// TIA Portal project "Tunel_Perozovodsk_2000_V3(LowSensorWater)" (V16)

(* hardware
DEVICE "S7-1200 station_1"  S7-1200 Station
   slot 0: "Rack_0"  S7-1200 Rack  Rack  V1.0
   slot 1: "PLC_Start"  CPU 1214C DC/DC/Rly  6ES7 214-1HG40-0XB0  V4.4
   slot 2: "DI 16x24VDC_1"  SM 1221 DI16 x 24VDC  6ES7 221-1BH30-0XB0  V1.0
   slot 3: "DQ 16xRelay_1"  SM 1222 DQ16 x relay  6ES7 222-1HH32-0XB0  V2.0
   slot 4: "AI 8xRTD_1"  SM 1231 AI8 x RTD  6ES7 231-5PF32-0XB0  V2.0
   slot 5: "AQ 4x14BIT_1"  6ES7 232-4HD32-0XB0  V2.1
   slot 6: "AQ 4x14BIT_2"  6ES7 232-4HD32-0XB0  V2.1
*)

// ===== PLC "PLC_Start"  CPU 1214C DC/DC/Rly =====

VAR_GLOBAL   // PLC tag table "Default tag table"
   "rAlarm_SetMinPressSteam" AT %MW12 : Int;   // Уставка минимального давления пара
   "rAI_Press1" AT %MW14 : Int;   // Давление датчика
   "bAlarmPress1" AT %M16.0 : Bool;
   "rAlarm_SetMinPressWater" AT %MW18 : Int;   // Уставка аварийного давления воды
   "rAI_Press2" AT %MW20 : Int;
   "test_PID_P_Backup" AT %MD28 : Real;
   "testLoadBackUp" AT %M1.1 : Bool;
   "Test_eee" AT %M1.2 : Bool;
END_VAR

VAR_GLOBAL   // PLC tag table "HMI_"
   "bHMI_button_Start" AT %M2.0 : Bool;   // Кнопка старт
   "bHMI_button_Stop" AT %M2.1 : Bool;   // Кнопка стоп
   "bHMI_button_Pause" AT %M2.2 : Bool;   // Кнопка пауза
   "bHMI_Button_ConveyorStart" AT %M2.4 : Bool;   // Кнопка подтверждения старта конвейера
   "bStartAllowed" AT %M100.0 : Bool;   // Готовность к старту
   "bOpenWindStartConveyor" AT %M100.1 : Bool;   // Вызов окна подтверждения оператором старта конвейера
   "iHMI_Num_StatrPaster" AT %MW4 : Int;   // Статус работы пастризаора
   "sHMI_Text_State" AT %MB3 : Char;   // Ткстом статус пастеризатора
   "bTypePID_Zone1" AT %M8.0 : Bool;   // Тип ПИД - 1 - Охлаждение, 0 - Нагрев
   "bTypePID_Zone2" AT %M8.1 : Bool;   // Тип ПИД - 1 - Охлаждение, 0 - Нагрев
   "bTypePID_Zone3" AT %M8.2 : Bool;   // Тип ПИД - 1 - Охлаждение, 0 - Нагрев
   "bTypePID_Zone4" AT %M8.3 : Bool;   // Тип ПИД - 1 - Охлаждение, 0 - Нагрев
   "bTypePID_Zone5" AT %M8.4 : Bool;   // Тип ПИД - 1 - Охлаждение, 0 - Нагрев
   "rHMI_SpeedConveyor" AT %MD60 : Real;   // Скорость конвейера
   "rHMI_TimeHoldMin" AT %MD56 : Real;   // Для удобства восприятия времени выдержки
   "bResetCommon" AT %M0.3 : Bool;   // Глобальный сброс аварий
   "bAllAuto" AT %M0.6 : Bool;   // Перевод всего оборудования в авто с ручного
   "bZoomerOff" AT %M0.7 : Bool;   // Выкл пищалка
   "bHMI_button_Start_Sterilization" AT %M2.5 : Bool;   // Кнопка старт Стерилизации
   "bHMI_Steril_Fimish" AT %M8.7 : Bool;   // Стерилизация готова флаг
   "iHMI_Steril_sec" AT %MW22 : Int;   // СЕК таймера стерилизациии
   "iHMI_Steril_min" AT %MW26 : Int;   // МИН таймера стерилизации
   "iHMIWind_FinishStiril" AT %MW32 : Int;   // Всплывающее окно на панели
   "bOpenWindSterilFinish" AT %M34.0 : Bool;   // Вызвать окно окончание стирилизации
END_VAR

VAR_GLOBAL   // PLC tag table "DI"
   "+Кнопка экстренной остановки E-Stop №1" AT %I0.0 : Bool;
   "+Кнопка экстренной остановки E-Stop №2" AT %I0.1 : Bool;
   "+Кнопка экстренной остановки E-Stop №3" AT %I0.2 : Bool;
   "+Реле напряжения и фаз. Напряжение в норма" AT %I3.0 : Bool;
   "+Датчик уровня 1 – нижний уровень" AT %I3.1 : Bool;
   "+Датчик уровня 1 – верхний уровень" AT %I3.2 : Bool;
   "+Индуктивный датчик конвейера 1" AT %I3.3 : Bool;
   "+Преобразователь частоты готов (работа) 1" AT %I3.4 : Bool;
   "+Преобразователь частоты готов (работа) 2" AT %I3.5 : Bool;
   "+Преобразователь частоты готов (работа) 3" AT %I3.6 : Bool;
   "+Мотор-автомат 1" AT %I0.3 : Bool;
   "+Мотор-автомат 2" AT %I0.4 : Bool;
   "Мотор-автомат 3" AT %I0.5 : Bool;
   "Мотор-автомат 4" AT %I0.6 : Bool;
   "Мотор-автомат 5" AT %I0.7 : Bool;
   "Мотор-автомат 6" AT %I1.0 : Bool;
   "Мотор-автомат 7" AT %I1.1 : Bool;
   "Мотор-автомат 8" AT %I1.2 : Bool;
   "+Мотор-автомат 9" AT %I1.3 : Bool;
   "+Мотор-автомат 10" AT %I1.4 : Bool;
   "+Пускатель включен 1" AT %I2.0 : Bool;
   "Пускатель включен 2" AT %I2.1 : Bool;
   "Пускатель включен 3" AT %I2.2 : Bool;
   "Пускатель включен 4" AT %I2.3 : Bool;
   "Пускатель включен 5" AT %I2.4 : Bool;
   "Пускатель включен 6" AT %I2.5 : Bool;
   "+Мотор-автомат 11" AT %I1.5 : Bool;
   "Пускатель включен 7" AT %I2.6 : Bool;
   "+Пускатель включен 8" AT %I2.7 : Bool;
END_VAR

VAR_GLOBAL   // PLC tag table "MyTags"
   "rHoldtimeMIN_Out" AT %MD52 : Real;   // Время выдержки в мин
   "Разрешение работы конвейера" AT %M0.0 : Bool;   // Команда разрешения от Глобального блока работы
   "Авария, ошибка в системе" AT %M0.1 : Bool;   // Метка ошибок или аварий
   "iNomberZoneAlarm" AT %MW6 : Int;   // Номер зоны с отклонениями
   "bMain_AlarmSystem" AT %M2.3 : Bool;   // АВария в системе (Общая)
   "bStartWork_Main_TunelPaster" AT %M1.7 : Bool;   // Старт-Работа тунельного пастеризатора (ОБЩИЙ)
   "bHasPrior_Stop" AT %M10.1 : Bool;   // Имеется маркер разрешения "СТОП - конвейер
   "bStateZones_OK" AT %M10.0 : Bool;   // Все зоны готовы к работе
   "bStartFillBac_1" AT %M0.4 : Bool;   // Ком_Наполнение бака 1
   "bStartFillBac_2" AT %M0.5 : Bool;   // Ком_Наполнение бака 2
   "AlarmPress" AT %M0.2 : Bool;   // Общая авария давления
   "bStartWork_Sterilization" AT %M2.6 : Bool;   // Старт-Работа режима стерилизации
   "bState_Stiril_Zone_OK" AT %M1.0 : Bool;   // Все зоны готовы к стерилизации
   "iNumZoneStiril_NotOk" AT %MW24 : Int;   // Номер зоны не готовые стирилизации
END_VAR

VAR_GLOBAL   // PLC tag table "Timers_CPU"
   "Time_0.1s" AT %M500.0 : Bool;
   "Time_0.2s" AT %M500.1 : Bool;
   "Time_0.4s" AT %M500.2 : Bool;
   "Time_0.5s" AT %M500.3 : Bool;
   "Time_0.8s" AT %M500.4 : Bool;
   "Time_1s" AT %M500.5 : Bool;
   "Time_1.6s" AT %M500.6 : Bool;
   "Time_2s" AT %M500.7 : Bool;
END_VAR

VAR_GLOBAL   // PLC tag table "DO"
   "Пневмо_остров клапан 1" AT %Q0.0 : Bool;
   "Пневмо_остров клапан 2" AT %Q0.1 : Bool;
   "Пневмо_остров клапан 3" AT %Q0.2 : Bool;
   "Пневмо_остров клапан 4" AT %Q0.3 : Bool;
   "Пневмо_остров клапан 5" AT %Q0.4 : Bool;
   "Пневмо_остров клапан 6" AT %Q0.5 : Bool;
   "Пневмо_остров клапан 7" AT %Q0.6 : Bool;
   "Пневмо_остров клапан 8" AT %Q0.7 : Bool;
   "Пневмо_остров клапан 9" AT %Q1.0 : Bool;
   "Пневмо_остров клапан 10" AT %Q1.1 : Bool;
   "Преобразователь частоты - пуск 1" AT %Q4.0 : Bool;   // Реле К 9
   "Преобразователь частоты - пуск 2" AT %Q4.1 : Bool;   // Реле К 10
   "Преобразователь частоты - пуск 3" AT %Q4.2 : Bool;   // Реле К 11
   "Световая колонна - зеленый" AT %Q4.6 : Bool;
   "Световая колонна - желтый" AT %Q4.5 : Bool;
   "Световая колонна - красный" AT %Q4.4 : Bool;
   "Световая колонна – звуковой сигнал" AT %Q4.7 : Bool;
   "Пускатель №1" AT %Q5.0 : Bool;
   "Пускатель №2" AT %Q5.1 : Bool;
   "Пускатель №3" AT %Q5.2 : Bool;
   "Пускатель №4" AT %Q5.3 : Bool;
   "Пускатель №5" AT %Q5.4 : Bool;
   "Пускатель №6" AT %Q5.5 : Bool;
   "Пускатель №7" AT %Q5.6 : Bool;
   "Пускатель Воздуходувка" AT %Q5.7 : Bool;
   "Пуск транспортера" AT %Q4.3 : Bool;   // Реле К 12
END_VAR

VAR_GLOBAL   // PLC tag table "AI"
   "Датчик температуры 1" AT %IW140 : Int;   // PT100
   "Датчик температуры 2" AT %IW142 : Int;   // PT100
   "Датчик температуры 3" AT %IW144 : Int;   // PT100
   "Датчик температуры 4" AT %IW146 : Int;   // PT100
   "Датчик температуры 5" AT %IW148 : Int;   // PT100
   "Датчик температуры 6" AT %IW150 : Int;   // PT100
   "Датчик температуры 7" AT %IW152 : Int;   // PT100
   "AI_0.7_" AT %IW174 : Int;   // PT100
   "AI_0.0_Датчик давления 1" AT %IW112 : Int;   // 4-20mA
   "AI_0.1_Датчик давления 2" AT %IW114 : Int;   // 4-20mA
   "AI_0.2_Датчик давления 3" AT %IW116 : Int;   // 4-20mA
   "AI_0.3_" AT %IW118 : Int;   // 4-20mA
END_VAR

VAR_GLOBAL   // PLC tag table "AO"
   "Преобразователь частоты 1" AT %QW182 : Int;
   "Преобразователь частоты 2" AT %QW184 : Int;
   "Преобразователь частоты 3" AT %QW186 : Int;
   "Преобразователь частоты 4" AT %QW190 : Int;
   "Управляемый клапан №1" AT %QW160 : Int;
   "Управляемый клапан №2" AT %QW162 : Int;
   "Управляемый клапан №3" AT %QW164 : Int;
   "Управляемый клапан №4" AT %QW166 : Int;
   "Управляемый клапан №5" AT %QW180 : Int;
END_VAR

VAR_GLOBAL   // PLC tag table "Alarms"
   "Ai_Alarm_1" AT %M50.0 : Bool;
   "Ai_Alarm_2" AT %M50.1 : Bool;
   "Ai_Alarm_3" AT %M50.2 : Bool;
   "Ai_Alarm_4" AT %M50.3 : Bool;
   "Ai_Alarm_5" AT %M50.4 : Bool;
   "Ai_Alarm_6" AT %M50.5 : Bool;
END_VAR

VAR_GLOBAL   // PLC tag table "__TEST"
   "bT_Alarm" AT %M1.3 : Bool;
   "bTOpenWind" AT %M1.4 : Bool;
   "iTestPause" AT %MW1 : Int;
   "bTZoomOff" AT %M8.5 : Bool;
END_VAR

TYPE "FV_o/c"
   STRUCT
      bOpenCmd : Bool;   // Команда открыть (автомат)
      bManualMode : Bool;   // Ручной режим (TRUE)
      bManualOpen : Bool;   // Команда открыть в ручном режиме
      bFeedbackOpen : Bool;   // Обратная связь "Открыт"
      tMaxTime : Time;   // Время на открытие
      bResetAlarm : Bool;   // Сброс аварии
      bCheckFeedback : Bool;   // Выбирается есть ли обратная связь у клапана
      bOutOpen : Bool;   // Выход на открытие клапана
      iOutState : Int;   // Выход статуса клапана
   END_STRUCT;
END_TYPE

TYPE "ZoneStatus"
   STRUCT
      bInSetpoint : Bool;   // Зона в уставке по температуре
      bOutOfRange : Bool;   // Зона вышла от уставки на > дельта
      bHasPriority : Bool;   // Зона имеет приоритет на остановку конвейера
   END_STRUCT;
END_TYPE

TYPE "Zone_Pararm"
   STRUCT
      rTemp : Real;   // Температура с датчика
      rSet : Real := 20.0;   // Уставка
      rDeltaDown : Real := 1.0;   // ДельтаНижний предел
      rDeltaUP : Real := 1.0;   // ДельтаВерхний Предел
      bPriority : Bool;   // Приоритет
      bOUT_ZoneStatus : "ZoneStatus";   // Состояние зоны_
   END_STRUCT;
END_TYPE

TYPE "FV_regul"
   STRUCT
      bHMI_ManualMode : Bool;   // Переключение режима авто/ручно (0 - А, 1 - Р)
      "bManualOpen/Close" : Bool;   // Ручн режим выход DO для клапана
      rHMI_ManualSet : Real;   // Уставка в ручном режиме (0-100)
      "bAutoOpen/Close" : Bool;   // Авто режим Сигнал DO на выход для клапана
      rAuto_Set : Real;   // Уставка в автоматическом режиме
      iOut_AO : Int;   // Сигнал на аналоговый выход
      "rHMI_Out_FV-%" : Real;   // Состояние в % (0-100)
      "bOut_DO_Open/Close" : Bool;   // Сигнал выход для DO
      bOut_State_ValveOpen : Int;   // Cтатуса - клапан открыт (1)/закрыт(0)
   END_STRUCT;
END_TYPE

TYPE "Коэф ПИД"
   STRUCT
      Set : Real;   // Уставка
      Gain : Int;   // Коэф П
      I : DInt;   // Коэф И
      D : DInt;   // Коэф Д
   END_STRUCT;
END_TYPE

TYPE "PE_Param"
   STRUCT
      rПЕ_Задан : Real;
      rДлина_Конв : Real;
      rZ_Коэф : Real := 1.393;
      rТref : Real := 60.0;
      rТемп_Мин : Real;
      rТемп_Макс : Real;
      "rСкоростьКонв_м/мин" : Real;
      rРучноеЗначТемп : Real;
      diВремяПростоя : DInt := 60000;
      bManualTemp : Bool;
   END_STRUCT;
END_TYPE

TYPE "tipe_Pumps"
   STRUCT
      bAutoMode_Work : Bool;   // автоматический режим
      bManualMode : Bool;   // Ручной режим вкл/выкл
      bManualStart : Bool;   // Старт в ручном режиме
      rManualSpeed : Real;   // Скорость в ручном режиме
      rHMI_Speed : Real;   // Выходная скороость для HMI
      bHMI_PumpRun : Bool;   // Статус работы для HMI
      bresAlarm : Bool;   // Сброс аварий
      iStatusPump : Int;   // Статус насоса
      bIn_DryRunning : Bool;   // Сигнал сухого хода
      bIn_AutomatState : Bool;   // Вход статуса состояния автоматов
      bIn_PuskatelState : Bool;   // Вход статуса состояния пускателя
      bIn_Run_Ok_State : Bool;   // Вход подтверждения старта (частотники)
   END_STRUCT;
END_TYPE

TYPE "Tipe_Conveyor"
   STRUCT
      bManualMode : Bool;   // Ручной режим вкл/выкл
      bManualStart : Bool;   // Старт в ручном режиме
      rManualSpeed : Real;   // Скорость в ручном режиме
      bresAlarm : Bool;   // Сброс аварий
      rAutoSpeed : Real;   // Автомат_Заданная скорость конвеера
      rHMI_Speed : Real;   // Выходная скороость для HMI
      bHMI_Conv_Run : Bool;   // Статус работы для HMI
      iStatusConve : Int;   // Статус конвейера
      bIn_AutomatState : Bool;   // Вход статуса состояния автоматов
      bInPuskatelState : Bool;   // Вход статуса состояния пускателя
      bInRun_Ok_State : Bool;   // Вход подтверждения старта (частотники)
   END_STRUCT;
END_TYPE

TYPE "Tipe_DI"
   STRUCT
      f_DI_out : Bool;
      "bFiltr_on/off" : Bool := true;   // Вкл/выкл фильтрацию входа
      diTime_filtr : Time := T#100ms;   // Уставка времени фильтрации
      bSimulation : Bool;   // Включение режима симуляции
      "bSim_On/Off" : Bool;   // Управление симуляцией
   END_STRUCT;
END_TYPE

TYPE "Tipe_Filling_Bac"
   STRUCT
      bManualMode : Bool;
      bManualOpen : Bool;
      diTimeCloseValve : DInt;   // Таймер задержки закрытия клапана по верхнему уровню
   END_STRUCT;
END_TYPE

TYPE "Tipe_AI"
   STRUCT
      bSimulate : Bool;   // Вкл симуляции датчика
      rSimulateValue : Real;   // Значение симуляции датчика
      rSensor_HL : Real;   // Верхний предел датчика
      rSensor_LL : Real;   // Нижний предел датчика
      bFiltr : Bool;   // Управление фильтром значений
      rAI_Value : Real;   // Значение аналогового датчика
   END_STRUCT;
END_TYPE

TYPE "tipePress"
   STRUCT
      rInPress : Real;   // Значение с датчика
      rSetpoint : Real := 2.0;   // Уставка минимального давления
      bAlarm_Press : Bool;   // Выход АВАРИЯ
   END_STRUCT;
END_TYPE

DATA_BLOCK "Test_Beep_DB"   // DB129
{ S7_Optimized_Access := 'TRUE' }
VERSION : 0.1
// stored: InstanceOfName Test_Beep
"Test_Beep"
BEGIN
END_DATA_BLOCK

// folder: AI_Signal/AI_DB/PT100

DATA_BLOCK "AI_1_(PT100)_DB"   // DB88
{ S7_Optimized_Access := 'FALSE' }
VERSION : 0.1
// stored: InstanceOfName AI_(PT100)
"AI_(PT100)"
BEGIN
END_DATA_BLOCK

DATA_BLOCK "AI_2_(PT100)_DB"   // DB89
{ S7_Optimized_Access := 'FALSE' }
VERSION : 0.1
// stored: InstanceOfName AI_(PT100)
"AI_(PT100)"
BEGIN
END_DATA_BLOCK

DATA_BLOCK "AI_3_(PT100)_DB"   // DB91
{ S7_Optimized_Access := 'FALSE' }
VERSION : 0.1
// stored: InstanceOfName AI_(PT100)
"AI_(PT100)"
BEGIN
END_DATA_BLOCK

DATA_BLOCK "AI_4_(PT100)_DB"   // DB92
{ S7_Optimized_Access := 'FALSE' }
VERSION : 0.1
// stored: InstanceOfName AI_(PT100)
"AI_(PT100)"
BEGIN
END_DATA_BLOCK

DATA_BLOCK "AI_5_(PT100)_DB"   // DB93
{ S7_Optimized_Access := 'FALSE' }
VERSION : 0.1
// stored: InstanceOfName AI_(PT100)
"AI_(PT100)"
BEGIN
END_DATA_BLOCK

DATA_BLOCK "AI_6_(PT100)_DB"   // DB112
{ S7_Optimized_Access := 'FALSE' }
VERSION : 0.1
// stored: InstanceOfName AI_(PT100)
"AI_(PT100)"
BEGIN
END_DATA_BLOCK

DATA_BLOCK "AI_7_(PT100)_DB"   // DB113
{ S7_Optimized_Access := 'FALSE' }
VERSION : 0.1
// stored: InstanceOfName AI_(PT100)
"AI_(PT100)"
BEGIN
END_DATA_BLOCK

// folder: DB-FB

DATA_BLOCK "FB_check_For_Start_DB"   // DB1
{ S7_Optimized_Access := 'FALSE' }
VERSION : 0.1
// stored: InstanceOfName FB_check_For_Start
"FB_check_For_Start"
BEGIN
END_DATA_BLOCK

DATA_BLOCK "FB_Emergency_DB"   // DB3
{ S7_Optimized_Access := 'FALSE' }
VERSION : 0.1
// stored: InstanceOfName FB_Аварии
"FB_Аварии"
BEGIN
END_DATA_BLOCK

DATA_BLOCK "FB_CheckZoneStatus_DB"   // DB11
{ S7_Optimized_Access := 'FALSE' }
VERSION : 0.1
// stored: InstanceOfName FB_CheckZoneStatus
"FB_CheckZoneStatus"
BEGIN
END_DATA_BLOCK

DATA_BLOCK "FB_Управление конвейером_DB"   // DB18
{ S7_Optimized_Access := 'FALSE' }
VERSION : 0.1
// stored: InstanceOfName FB_Управление конвейером
"FB_Управление конвейером"
BEGIN
END_DATA_BLOCK

DATA_BLOCK "FB_GlobalStateManager_DB"   // DB31
{ S7_Optimized_Access := 'FALSE' }
VERSION : 0.1
// stored: InstanceOfName FB_GlobalStateManager
"FB_GlobalStateManager"
BEGIN
END_DATA_BLOCK

DATA_BLOCK "FB_PE_Control_DB"   // DB38
{ S7_Optimized_Access := 'TRUE' }
VERSION : 0.1
// stored: InstanceOfName FB_ПЕ_Control
"FB_ПЕ_Control"
BEGIN
END_DATA_BLOCK

DATA_BLOCK "Главный блок конвейера_DB"   // DB39
{ S7_Optimized_Access := 'TRUE' }
VERSION : 0.1
// stored: InstanceOfName FB_Главный блок конвейера
"FB_Главный блок конвейера"
BEGIN
END_DATA_BLOCK

DATA_BLOCK "R_trig_All_Auto"   // DB40
{ S7_Optimized_Access := 'TRUE' }
VERSION : 0.1
// stored: InstanceOfName R_trig
"R_trig"
BEGIN
END_DATA_BLOCK

DATA_BLOCK "FB_Sterilization_CheckZoneStatus_DB"   // DB41
{ S7_Optimized_Access := 'FALSE' }
VERSION : 0.1
// stored: InstanceOfName FB_Stiril_CheckZoneStatus
"FB_Stiril_CheckZoneStatus"
BEGIN
END_DATA_BLOCK

DATA_BLOCK "FB_Steril_Timer_DB"   // DB42
{ S7_Optimized_Access := 'TRUE' }
VERSION : 0.1
// stored: InstanceOfName FB_Steril_Timer
"FB_Steril_Timer"
BEGIN
END_DATA_BLOCK

DATA_BLOCK "Вентилятор_DB"   // DB46
{ S7_Optimized_Access := 'FALSE' }
VERSION : 0.1
// stored: InstanceOfName Pump
"Pump"
BEGIN
END_DATA_BLOCK

DATA_BLOCK "FB_Mode_Paster_DB"   // DB81
{ S7_Optimized_Access := 'TRUE' }
VERSION : 0.1
// stored: InstanceOfName FB_Mode_Paster
"FB_Mode_Paster"
BEGIN
END_DATA_BLOCK

DATA_BLOCK "FB_Filling_Bac1_DB"   // DB84
{ S7_Optimized_Access := 'TRUE' }
VERSION : 0.1
// stored: InstanceOfName FB_Filling_Bac
"FB_Filling_Bac"
BEGIN
END_DATA_BLOCK

DATA_BLOCK "FB_Filling_Bac2_DB"   // DB86
{ S7_Optimized_Access := 'TRUE' }
VERSION : 0.1
// stored: InstanceOfName FB_Filling_Bac
"FB_Filling_Bac"
BEGIN
END_DATA_BLOCK

DATA_BLOCK "FB_Press_Controll_Water_DB"   // DB96
{ S7_Optimized_Access := 'TRUE' }
VERSION : 0.1
// stored: InstanceOfName FB_Press_Controll
"FB_Press_Controll"
BEGIN
END_DATA_BLOCK

DATA_BLOCK "FB_Press_Controll_Steam_DB"   // DB97
{ S7_Optimized_Access := 'TRUE' }
VERSION : 0.1
// stored: InstanceOfName FB_Press_Controll
"FB_Press_Controll"
BEGIN
END_DATA_BLOCK

DATA_BLOCK "FB_Press_Controll_Glikol_DB"   // DB98
{ S7_Optimized_Access := 'TRUE' }
VERSION : 0.1
// stored: InstanceOfName FB_Press_Controll
"FB_Press_Controll"
BEGIN
END_DATA_BLOCK

DATA_BLOCK "R_trig_DB"   // DB99
{ S7_Optimized_Access := 'TRUE' }
VERSION : 0.1
// stored: InstanceOfName R_trig
"R_trig"
BEGIN
END_DATA_BLOCK

DATA_BLOCK "R_trig_DB_Alarm_Zoomer"   // DB101
{ S7_Optimized_Access := 'TRUE' }
VERSION : 0.1
// stored: InstanceOfName R_trig
"R_trig"
BEGIN
END_DATA_BLOCK

DATA_BLOCK "FB_SVETOFOR_DB"   // DB102
{ S7_Optimized_Access := 'TRUE' }
VERSION : 0.1
// stored: InstanceOfName FB_SVETOFOR
"FB_SVETOFOR"
BEGIN
END_DATA_BLOCK

DATA_BLOCK "FB_check_For_StartSterilization_DB"   // DB103
{ S7_Optimized_Access := 'FALSE' }
VERSION : 0.1
// stored: InstanceOfName FB_check_For_Start
"FB_check_For_Start"
BEGIN
END_DATA_BLOCK

DATA_BLOCK "FB_STIRIL_Mode_DB"   // DB115
{ S7_Optimized_Access := 'TRUE' }
VERSION : 0.1
// stored: InstanceOfName FB_Mode_STIRIL
"FB_Mode_STIRIL"
BEGIN
END_DATA_BLOCK

DATA_BLOCK "R_trig_OpenWindOper"   // DB124
{ S7_Optimized_Access := 'TRUE' }
VERSION : 0.1
// stored: InstanceOfName R_trig
"R_trig"
BEGIN
END_DATA_BLOCK

DATA_BLOCK "R_trig_Puasa"   // DB125
{ S7_Optimized_Access := 'TRUE' }
VERSION : 0.1
// stored: InstanceOfName R_trig
"R_trig"
BEGIN
END_DATA_BLOCK

// folder: DI_signal/DB_DI

DATA_BLOCK "DI_EStop1"   // DB48
{ S7_Optimized_Access := 'FALSE' }
VERSION : 0.1
// stored: InstanceOfName FB_DI
"FB_DI"
BEGIN
END_DATA_BLOCK

DATA_BLOCK "DI_EStop2"   // DB49
{ S7_Optimized_Access := 'FALSE' }
VERSION : 0.1
// stored: InstanceOfName FB_DI
"FB_DI"
BEGIN
END_DATA_BLOCK

DATA_BLOCK "DI_EStop3"   // DB50
{ S7_Optimized_Access := 'FALSE' }
VERSION : 0.1
// stored: InstanceOfName FB_DI
"FB_DI"
BEGIN
END_DATA_BLOCK

DATA_BLOCK "DI_ReleVolt"   // DB51
{ S7_Optimized_Access := 'FALSE' }
VERSION : 0.1
// stored: InstanceOfName FB_DI
"FB_DI"
BEGIN
END_DATA_BLOCK

DATA_BLOCK "DI_1_Уровень_Низ"   // DB52
{ S7_Optimized_Access := 'FALSE' }
VERSION : 0.1
// stored: InstanceOfName FB_DI
"FB_DI"
BEGIN
END_DATA_BLOCK

DATA_BLOCK "DI_1_Уровень_Верх"   // DB53
{ S7_Optimized_Access := 'FALSE' }
VERSION : 0.1
// stored: InstanceOfName FB_DI
"FB_DI"
BEGIN
END_DATA_BLOCK

DATA_BLOCK "DI_2_Уровень_Низ"   // DB54
{ S7_Optimized_Access := 'FALSE' }
VERSION : 0.1
// stored: InstanceOfName FB_DI
"FB_DI"
BEGIN
END_DATA_BLOCK

DATA_BLOCK "DI_2_Уровень_Верх"   // DB55
{ S7_Optimized_Access := 'FALSE' }
VERSION : 0.1
// stored: InstanceOfName FB_DI
"FB_DI"
BEGIN
END_DATA_BLOCK

DATA_BLOCK "DI_Индуктивный датчик конв - 1"   // DB56
{ S7_Optimized_Access := 'FALSE' }
VERSION : 0.1
// stored: InstanceOfName FB_DI
"FB_DI"
BEGIN
END_DATA_BLOCK

DATA_BLOCK "DI_Индуктивный датчик конв - 2"   // DB57
{ S7_Optimized_Access := 'FALSE' }
VERSION : 0.1
// stored: InstanceOfName FB_DI
"FB_DI"
BEGIN
END_DATA_BLOCK

DATA_BLOCK "DI_Частотник_1_Готов"   // DB58
{ S7_Optimized_Access := 'FALSE' }
VERSION : 0.1
// stored: InstanceOfName FB_DI
"FB_DI"
BEGIN
END_DATA_BLOCK

DATA_BLOCK "DI_Частотник_2_Готов"   // DB59
{ S7_Optimized_Access := 'FALSE' }
VERSION : 0.1
// stored: InstanceOfName FB_DI
"FB_DI"
BEGIN
END_DATA_BLOCK

DATA_BLOCK "DI_Частотник_3_Готов"   // DB60
{ S7_Optimized_Access := 'FALSE' }
VERSION : 0.1
// stored: InstanceOfName FB_DI
"FB_DI"
BEGIN
END_DATA_BLOCK

DATA_BLOCK "DI_Частотник_4_Готов"   // DB61
{ S7_Optimized_Access := 'FALSE' }
VERSION : 0.1
// stored: InstanceOfName FB_DI
"FB_DI"
BEGIN
END_DATA_BLOCK

DATA_BLOCK "DI_Мотор-Автомат-1(вкл)"   // DB62
{ S7_Optimized_Access := 'FALSE' }
VERSION : 0.1
// stored: InstanceOfName FB_DI
"FB_DI"
BEGIN
END_DATA_BLOCK

DATA_BLOCK "DI_Мотор-Автомат-2(вкл)"   // DB63
{ S7_Optimized_Access := 'FALSE' }
VERSION : 0.1
// stored: InstanceOfName FB_DI
"FB_DI"
BEGIN
END_DATA_BLOCK

DATA_BLOCK "DI_Мотор-Автомат-3(вкл)"   // DB64
{ S7_Optimized_Access := 'FALSE' }
VERSION : 0.1
// stored: InstanceOfName FB_DI
"FB_DI"
BEGIN
END_DATA_BLOCK

DATA_BLOCK "DI_Мотор-Автомат-4(вкл)"   // DB65
{ S7_Optimized_Access := 'FALSE' }
VERSION : 0.1
// stored: InstanceOfName FB_DI
"FB_DI"
BEGIN
END_DATA_BLOCK

DATA_BLOCK "DI_Мотор-Автомат-5(вкл)"   // DB66
{ S7_Optimized_Access := 'FALSE' }
VERSION : 0.1
// stored: InstanceOfName FB_DI
"FB_DI"
BEGIN
END_DATA_BLOCK

DATA_BLOCK "DI_Мотор-Автомат-6(вкл)"   // DB67
{ S7_Optimized_Access := 'FALSE' }
VERSION : 0.1
// stored: InstanceOfName FB_DI
"FB_DI"
BEGIN
END_DATA_BLOCK

DATA_BLOCK "DI_Мотор-Автомат-7(вкл)"   // DB68
{ S7_Optimized_Access := 'FALSE' }
VERSION : 0.1
// stored: InstanceOfName FB_DI
"FB_DI"
BEGIN
END_DATA_BLOCK

DATA_BLOCK "DI_Мотор-Автомат-8(вкл)"   // DB69
{ S7_Optimized_Access := 'FALSE' }
VERSION : 0.1
// stored: InstanceOfName FB_DI
"FB_DI"
BEGIN
END_DATA_BLOCK

DATA_BLOCK "DI_Мотор-Автомат-9(вкл)"   // DB70
{ S7_Optimized_Access := 'FALSE' }
VERSION : 0.1
// stored: InstanceOfName FB_DI
"FB_DI"
BEGIN
END_DATA_BLOCK

DATA_BLOCK "DI_Мотор-Автомат-10(вкл)"   // DB71
{ S7_Optimized_Access := 'FALSE' }
VERSION : 0.1
// stored: InstanceOfName FB_DI
"FB_DI"
BEGIN
END_DATA_BLOCK

DATA_BLOCK "DI_Пускатель - 1(вкл)"   // DB72
{ S7_Optimized_Access := 'FALSE' }
VERSION : 0.1
// stored: InstanceOfName FB_DI
"FB_DI"
BEGIN
END_DATA_BLOCK

DATA_BLOCK "DI_Пускатель - 2(вкл)"   // DB73
{ S7_Optimized_Access := 'FALSE' }
VERSION : 0.1
// stored: InstanceOfName FB_DI
"FB_DI"
BEGIN
END_DATA_BLOCK

DATA_BLOCK "DI_Пускатель - 3(вкл)"   // DB74
{ S7_Optimized_Access := 'FALSE' }
VERSION : 0.1
// stored: InstanceOfName FB_DI
"FB_DI"
BEGIN
END_DATA_BLOCK

DATA_BLOCK "DI_Пускатель - 4(вкл)"   // DB75
{ S7_Optimized_Access := 'FALSE' }
VERSION : 0.1
// stored: InstanceOfName FB_DI
"FB_DI"
BEGIN
END_DATA_BLOCK

DATA_BLOCK "DI_Пускатель - 5(вкл)"   // DB76
{ S7_Optimized_Access := 'FALSE' }
VERSION : 0.1
// stored: InstanceOfName FB_DI
"FB_DI"
BEGIN
END_DATA_BLOCK

DATA_BLOCK "DI_Пускатель - 6(вкл)"   // DB77
{ S7_Optimized_Access := 'FALSE' }
VERSION : 0.1
// stored: InstanceOfName FB_DI
"FB_DI"
BEGIN
END_DATA_BLOCK

DATA_BLOCK "DI_Мотор-Автомат-11(вкл)"   // DB116
{ S7_Optimized_Access := 'FALSE' }
VERSION : 0.1
// stored: InstanceOfName FB_DI
"FB_DI"
BEGIN
END_DATA_BLOCK

DATA_BLOCK "DI_Пускатель - 7(вкл)"   // DB117
{ S7_Optimized_Access := 'FALSE' }
VERSION : 0.1
// stored: InstanceOfName FB_DI
"FB_DI"
BEGIN
END_DATA_BLOCK

DATA_BLOCK "DI_Пускатель - 8(вкл)"   // DB118
{ S7_Optimized_Access := 'FALSE' }
VERSION : 0.1
// stored: InstanceOfName FB_DI
"FB_DI"
BEGIN
END_DATA_BLOCK

// folder: System blocks/Program resources

DATA_BLOCK "IEC_Timer_0_DB"   // DB44
{ S7_Optimized_Access := 'TRUE' }
AUTHOR : Simatic
FAMILY : IEC
NAME : IEC_TMR
VERSION : 1.0
// stored: InstanceOfName IEC_TIMER
"IEC_TIMER"
BEGIN
END_DATA_BLOCK

DATA_BLOCK "IEC_Timer_0_DB_1"   // DB45
{ S7_Optimized_Access := 'TRUE' }
AUTHOR : Simatic
FAMILY : IEC
NAME : IEC_TMR
VERSION : 1.0
// stored: InstanceOfName IEC_TIMER
"IEC_TIMER"
BEGIN
END_DATA_BLOCK

DATA_BLOCK "IEC_Timer_0_DB_3"   // DB47
{ S7_Optimized_Access := 'TRUE' }
AUTHOR : Simatic
FAMILY : IEC
NAME : IEC_TMR
VERSION : 1.0
// stored: InstanceOfName IEC_TIMER
"IEC_TIMER"
BEGIN
END_DATA_BLOCK

DATA_BLOCK "IEC_Timer_0_DB_2"   // DB100
{ S7_Optimized_Access := 'TRUE' }
AUTHOR : Simatic
FAMILY : IEC
NAME : IEC_TMR
VERSION : 1.0
// stored: InstanceOfName IEC_TIMER
"IEC_TIMER"
BEGIN
END_DATA_BLOCK

DATA_BLOCK "IEC_Timer_0_DB_4"   // DB120
{ S7_Optimized_Access := 'TRUE' }
AUTHOR : Simatic
FAMILY : IEC
NAME : IEC_TMR
VERSION : 1.0
// stored: InstanceOfName IEC_TIMER
"IEC_TIMER"
BEGIN
END_DATA_BLOCK

DATA_BLOCK "IEC_Timer_0_DB_5"   // DB121
{ S7_Optimized_Access := 'TRUE' }
AUTHOR : Simatic
FAMILY : IEC
NAME : IEC_TMR
VERSION : 1.0
// stored: InstanceOfName IEC_TIMER
"IEC_TIMER"
BEGIN
END_DATA_BLOCK

DATA_BLOCK "IEC_Timer_0_DB_10"   // DB122
{ S7_Optimized_Access := 'TRUE' }
AUTHOR : Simatic
FAMILY : IEC
NAME : IEC_TMR
VERSION : 1.0
// stored: InstanceOfName IEC_TIMER
"IEC_TIMER"
BEGIN
END_DATA_BLOCK

DATA_BLOCK "IEC_Timer_0_DB_11"   // DB123
{ S7_Optimized_Access := 'TRUE' }
AUTHOR : Simatic
FAMILY : IEC
NAME : IEC_TMR
VERSION : 1.0
// stored: InstanceOfName IEC_TIMER
"IEC_TIMER"
BEGIN
END_DATA_BLOCK

// folder: Use VARs to HMI

DATA_BLOCK "DB2_HMI_SET"   // DB2
{ S7_Optimized_Access := 'FALSE' }
VERSION : 0.1
   VAR
      dwSetMinWaitGoPause : DInt := 1;   // Время ожидания при выходе за пределы уставок
      dwSetMinWaitComeToGo : DInt := 1;   // Время ожидания при возврате к уставкам
      dwSetTimeWaitToStart : DInt := 60;   // Время ожидания выхода на режим пастеризатора
      dwSetTimeWaitToSPause : DInt := 60;   // Время ожидания Нахождения в паузе
      k_PID_Zona1 : "Коэф ПИД";   // ПИД - ЗОна 1
      k_PID_Zona2 : "Коэф ПИД";   // ПИД - зона 2
      k_PID_Zona3 : "Коэф ПИД";   // ПИД - ЗОна 3
      k_PID_Zona4 : "Коэф ПИД";   // ПИД - зона 4
      k_PID_Zona7 : "Коэф ПИД";   // ПИД - ЗОна 7
      HMI_PE : "PE_Param";
      iTime_Steriliz : Int := 10;   // Время стерилизации
   END_VAR
BEGIN
   k_PID_Zona1.Gain := 1;
   k_PID_Zona1.I := 20;
   k_PID_Zona2.Gain := 1;
   k_PID_Zona2.I := 20;
   k_PID_Zona3.Gain := 1;
   k_PID_Zona3.I := 20;
   k_PID_Zona4.Gain := 1;
   k_PID_Zona4.I := 20;
   k_PID_Zona7.Gain := 1;
   k_PID_Zona7.I := 20;
   HMI_PE.rПЕ_Задан := 65.0;
   HMI_PE.rДлина_Конв := 2.1;
   HMI_PE.rТемп_Макс := 100.0;
   HMI_PE."rСкоростьКонв_м/мин" := 0.24;
   HMI_PE.diВремяПростоя := 900000;
END_DATA_BLOCK

DATA_BLOCK "FVs_o/p"   // DB6
{ S7_Optimized_Access := 'FALSE' }
VERSION : 0.1
   VAR
      FV_1 : "FV_o/c";   // Подпитка
      FV_2 : "FV_o/c";   // Пар
      FV_3 : "FV_o/c";   // Стерилизация
   END_VAR
BEGIN
END_DATA_BLOCK

DATA_BLOCK "ЗОНЫ_Параметры"   // DB15
{ S7_Optimized_Access := 'FALSE' }
VERSION : 0.1
   VAR
      Zone_1 : "Zone_Pararm";
      Zone_2 : "Zone_Pararm";
      Zone_3 : "Zone_Pararm";
      Zone_4 : "Zone_Pararm";
      Zone_5 : "Zone_Pararm";
      Zone_6 : "Zone_Pararm";
      Zone_7 : "Zone_Pararm";
   END_VAR
BEGIN
   Zone_1.rSet := 30.0;
   Zone_2.rTemp := 0.0;
   Zone_5.rTemp := 0.0;
   Zone_1.rDeltaDown := 3.0;
   Zone_2.rDeltaDown := 3.0;
   Zone_3.rDeltaDown := 3.0;
   Zone_5.rDeltaDown := 3.0;
   Zone_2.rSet := 60.0;
   Zone_5.rSet := 20.0;
   Zone_3.bPriority := true;
END_DATA_BLOCK

DATA_BLOCK "FVs_Regul"   // DB24
{ S7_Optimized_Access := 'FALSE' }
VERSION : 0.1
   VAR
      FV_Regul_1 : "FV_regul";
      FV_Regul_2 : "FV_regul";
      FV_Regul_3 : "FV_regul";
      FV_Regul_4 : "FV_regul";
      FV_Regul_7 : "FV_regul";
   END_VAR
BEGIN
END_DATA_BLOCK

DATA_BLOCK "Pumps"   // DB30
{ S7_Optimized_Access := 'FALSE' }
VERSION : 0.1
   VAR
      Pump_1 : "tipe_Pumps";
      Pump_2 : "tipe_Pumps";
      Pump_3 : "tipe_Pumps";
      Pump_4 : "tipe_Pumps";
      Pump_5 : "tipe_Pumps";
      Pump_6 : "tipe_Pumps";
      Pump_7 : "tipe_Pumps";
   END_VAR
BEGIN
END_DATA_BLOCK

DATA_BLOCK "DI"   // DB43
{ S7_Optimized_Access := 'FALSE' }
VERSION : 0.1
   VAR
      DI_0 : "Tipe_DI";
      DI_1 : "Tipe_DI";
      DI_2 : "Tipe_DI";
      DI_3 : "Tipe_DI";
      DI_4 : "Tipe_DI";
      DI_5 : "Tipe_DI";
      DI_6 : "Tipe_DI";
      DI_7 : "Tipe_DI";
      DI_8 : "Tipe_DI";
      DI_9 : "Tipe_DI";
      DI_10 : "Tipe_DI";
      DI_11 : "Tipe_DI";
      DI_12 : "Tipe_DI";
      DI_13 : "Tipe_DI";
      DI_14 : "Tipe_DI";
      DI_15 : "Tipe_DI";
      DI_16 : "Tipe_DI";
      DI_17 : "Tipe_DI";
      DI_18 : "Tipe_DI";
      DI_19 : "Tipe_DI";
      DI_20 : "Tipe_DI";
      DI_21 : "Tipe_DI";
      DI_22 : "Tipe_DI";
      DI_23 : "Tipe_DI";
      DI_24 : "Tipe_DI";
      DI_25 : "Tipe_DI";
      DI_26 : "Tipe_DI";
      DI_27 : "Tipe_DI";
      DI_28 : "Tipe_DI";
      DI_29 : "Tipe_DI";
      DI_30 : "Tipe_DI";
      DI_31 : "Tipe_DI";
   END_VAR
BEGIN
END_DATA_BLOCK

DATA_BLOCK "Conveyor"   // DB82
{ S7_Optimized_Access := 'FALSE' }
VERSION : 0.1
   VAR
      Conveyor_1 : "Tipe_Conveyor";
      Conveyor_2 : "Tipe_Conveyor";
      Conveyor_3 : "Tipe_Conveyor";
      Conveyor_4 : "Tipe_Conveyor";
   END_VAR
BEGIN
   Conveyor_1.rManualSpeed := 0.0;
   Conveyor_1.rAutoSpeed := 70.0;
   Conveyor_2.rAutoSpeed := 50.0;
   Conveyor_3.rAutoSpeed := 60.0;
   Conveyor_4.rAutoSpeed := 70.0;
END_DATA_BLOCK

DATA_BLOCK "Vent"   // DB83
{ S7_Optimized_Access := 'FALSE' }
VERSION : 0.1
   VAR
      Vent_1 : "tipe_Pumps";   // Вентилятор обдува
   END_VAR
BEGIN
END_DATA_BLOCK

DATA_BLOCK "Filling_BacLevel"   // DB85
{ S7_Optimized_Access := 'FALSE' }
VERSION : 0.1
   VAR
      "1" : "Tipe_Filling_Bac";   // 1 бак
   END_VAR
BEGIN
   "1".diTimeCloseValve := 5;
END_DATA_BLOCK

DATA_BLOCK "Alarms"   // DB87
{ S7_Optimized_Access := 'FALSE' }
VERSION : 0.1
   VAR
      Ai_Alarm : Array[1..7] of Struct   // Аварии датчиков аналоговых
         ALARM : Bool;
         RESET : Bool;
      END_STRUCT;
      Pump_Alarm : Array[1..7] of Struct   // Аварии насосов
         ALARM : Bool;
         RESET : Bool;
      END_STRUCT;
      Conveyor_Alarm : Array[1..4] of Struct   // Аварии конвейеров
         ALARM : Bool;
         RESET : Bool;
      END_STRUCT;
      Vent_Alarm : Struct   // Авария вентиляторов
         Vent_Alarm_1 : Bool;
         RESET : Bool;
      END_STRUCT;
      Avtomat_Off : Array[1..11] of Struct   // Контроль состояния вкл мотор автоматов
         ALARM : Bool;
      END_STRUCT;
      FV_Alarm : Array[1..7] of Struct   // Авария клапанов
         ALARM : Bool;
         RESET : Bool;
      END_STRUCT;
      "xE-Stop_1" : Bool;   // Авария по кнопке 1
      "xE-Stop_2" : Bool;   // Авария по кнопке 2
      "xE-Stop_3" : Bool;   // Авария по кнопке 3
      xVoltRele : Bool;   // Авария реле контроля фаз
      xSensorConveyorZator_1 : Bool;   // Авария затор на конвейере - 1
      xSensorConveyorZator_2 : Bool;   // Авария затор на конвейере - 2
      xLongPauseConv : Bool;   // Авария, долгое ожидание выхода конвейера из паузы
      xLongWaitZoneOk : Bool;   // Ааврия, долгий выход на уставки
   END_VAR
BEGIN
END_DATA_BLOCK

DATA_BLOCK "AI_DB"   // DB90
{ S7_Optimized_Access := 'FALSE' }
VERSION : 0.1
   VAR
      AI_1 : "Tipe_AI";
      AI_2 : "Tipe_AI";
      AI_3 : "Tipe_AI";
      AI_4 : "Tipe_AI";
      AI_5 : "Tipe_AI";
      AI_6 : "Tipe_AI";
      AI_7 : "Tipe_AI";
      "AI_4-20_1" : "Tipe_AI";   // Пар
      "AI_4-20_2" : "Tipe_AI";   // Вода
      "AI_4-20_3" : "Tipe_AI";   // Гликоль
   END_VAR
BEGIN
   "AI_4-20_1".rSensor_HL := 10.0;
   "AI_4-20_2".rSensor_HL := 10.0;
   "AI_4-20_3".rSensor_HL := 10.0;
   "AI_4-20_1".bFiltr := true;
   "AI_4-20_2".bFiltr := true;
   "AI_4-20_3".bFiltr := true;
   AI_1.bFiltr := true;
   AI_2.bFiltr := true;
   AI_3.bFiltr := true;
   AI_4.bFiltr := true;
   AI_5.bFiltr := true;
END_DATA_BLOCK

DATA_BLOCK "Control_Press_DB"   // DB95
{ S7_Optimized_Access := 'FALSE' }
VERSION : 0.1
   VAR
      PressWater : "tipePress";
      PressSteam : "tipePress";
      PressGlikol : "tipePress";
   END_VAR
BEGIN
   PressWater.rSetpoint := 0.0;
   PressSteam.rSetpoint := 0.0;
   PressGlikol.rSetpoint := 0.0;
END_DATA_BLOCK

DATA_BLOCK "Зоны_Стерилизации_Парам"   // DB104
{ S7_Optimized_Access := 'FALSE' }
VERSION : 0.1
   VAR
      "Steril_Zona-1" : "Zone_Pararm";   // параметры стерилизации зона-1
      "Steril_Zona-2" : "Zone_Pararm";   // параметры стерилизации зона-2
      "Steril_Zona-3" : "Zone_Pararm";   // параметры стерилизации зона-3
      "Steril_Zona-4" : "Zone_Pararm";   // параметры стерилизации зона-4
      "Steril_Zona-5" : "Zone_Pararm";   // параметры стерилизации зона-5
      "Steril_Zona-6" : "Zone_Pararm";   // параметры стерилизации зона-6
      "Steril_Zona-7" : "Zone_Pararm";   // параметры стерилизации зона-7
   END_VAR
BEGIN
END_DATA_BLOCK

DATA_BLOCK "My_VarS"   // DB119
{ S7_Optimized_Access := 'FALSE' }
VERSION : 0.1
   VAR
      b_Woter_LowLevel_T1 : Bool;   // Низкий Уровень воды Танк-1
      b_Woter_UpLewel_T1 : Bool;   // Верхний Уровень воды Танк-2
   END_VAR
BEGIN
END_DATA_BLOCK

// folder: Зоны/DB_Zone

DATA_BLOCK "FB_Zone_Control_1_DB"   // DB12
{ S7_Optimized_Access := 'FALSE' }
VERSION : 0.1
// stored: InstanceOfName FB_Zone_Control
"FB_Zone_Control"
BEGIN
END_DATA_BLOCK

DATA_BLOCK "FB_Zone_Control_2_DB"   // DB13
{ S7_Optimized_Access := 'FALSE' }
VERSION : 0.1
// stored: InstanceOfName FB_Zone_Control
"FB_Zone_Control"
BEGIN
END_DATA_BLOCK

DATA_BLOCK "FB_Zone_Control_3_DB"   // DB14
{ S7_Optimized_Access := 'FALSE' }
VERSION : 0.1
// stored: InstanceOfName FB_Zone_Control
"FB_Zone_Control"
BEGIN
END_DATA_BLOCK

DATA_BLOCK "FB_Zone_Control_4_DB"   // DB16
{ S7_Optimized_Access := 'FALSE' }
VERSION : 0.1
// stored: InstanceOfName FB_Zone_Control
"FB_Zone_Control"
BEGIN
END_DATA_BLOCK

DATA_BLOCK "FB_Zone_Control_5_DB"   // DB17
{ S7_Optimized_Access := 'FALSE' }
VERSION : 0.1
// stored: InstanceOfName FB_Zone_Control
"FB_Zone_Control"
BEGIN
END_DATA_BLOCK

DATA_BLOCK "FB_Zone_Control_7_DB"   // DB94
{ S7_Optimized_Access := 'FALSE' }
VERSION : 0.1
// stored: InstanceOfName FB_Zone_Control
"FB_Zone_Control"
BEGIN
END_DATA_BLOCK

DATA_BLOCK "FB_Zone_Control_6_DB"   // DB114
{ S7_Optimized_Access := 'FALSE' }
VERSION : 0.1
// stored: InstanceOfName FB_Zone_Control
"FB_Zone_Control"
BEGIN
END_DATA_BLOCK

// folder: Зоны/Стерилизация

DATA_BLOCK "FB_Zone_1_Control_Steriliz_DB"   // DB105
{ S7_Optimized_Access := 'FALSE' }
VERSION : 0.1
// stored: InstanceOfName FB_Zone_Control_Steriliz
"FB_Zone_Control_Steriliz"
BEGIN
END_DATA_BLOCK

DATA_BLOCK "FB_Zone_2_Control_Стерилизация_DB"   // DB106
{ S7_Optimized_Access := 'FALSE' }
VERSION : 0.1
// stored: InstanceOfName FB_Zone_Control_Steriliz
"FB_Zone_Control_Steriliz"
BEGIN
END_DATA_BLOCK

DATA_BLOCK "FB_Zone_3_Control_Стерилизация_DB"   // DB107
{ S7_Optimized_Access := 'FALSE' }
VERSION : 0.1
// stored: InstanceOfName FB_Zone_Control_Steriliz
"FB_Zone_Control_Steriliz"
BEGIN
END_DATA_BLOCK

DATA_BLOCK "FB_Zone_4_Control_Стерилизация_DB"   // DB108
{ S7_Optimized_Access := 'FALSE' }
VERSION : 0.1
// stored: InstanceOfName FB_Zone_Control_Steriliz
"FB_Zone_Control_Steriliz"
BEGIN
END_DATA_BLOCK

DATA_BLOCK "FB_Zone_5_Control_Стерилизация_DB"   // DB109
{ S7_Optimized_Access := 'FALSE' }
VERSION : 0.1
// stored: InstanceOfName FB_Zone_Control_Steriliz
"FB_Zone_Control_Steriliz"
BEGIN
END_DATA_BLOCK

DATA_BLOCK "FB_Zone_6_Control_Стерилизация_DB"   // DB110
{ S7_Optimized_Access := 'FALSE' }
VERSION : 0.1
// stored: InstanceOfName FB_Zone_Control_Steriliz
"FB_Zone_Control_Steriliz"
BEGIN
END_DATA_BLOCK

DATA_BLOCK "FB_Zone_7_Control_Стерилизация_DB"   // DB111
{ S7_Optimized_Access := 'FALSE' }
VERSION : 0.1
// stored: InstanceOfName FB_Zone_Control_Steriliz
"FB_Zone_Control_Steriliz"
BEGIN
END_DATA_BLOCK

// folder: Клапана/FV_o/C/FV_DB

DATA_BLOCK "FV_1"   // DB4
{ S7_Optimized_Access := 'FALSE' }
VERSION : 0.1
// stored: InstanceOfName Valve(c/o)
"Valve(c/o)"
BEGIN
END_DATA_BLOCK

DATA_BLOCK "FV_2"   // DB9
{ S7_Optimized_Access := 'FALSE' }
VERSION : 0.1
// stored: InstanceOfName Valve(c/o)
"Valve(c/o)"
BEGIN
END_DATA_BLOCK

DATA_BLOCK "FV_3"   // DB10
{ S7_Optimized_Access := 'FALSE' }
VERSION : 0.1
// stored: InstanceOfName Valve(c/o)
"Valve(c/o)"
BEGIN
END_DATA_BLOCK

// folder: Клапана/FV_regul/DB

DATA_BLOCK "FV_Regul_1_DB"   // DB20
{ S7_Optimized_Access := 'FALSE' }
VERSION : 0.1
// stored: InstanceOfName Valve(regul)
"Valve(regul)"
BEGIN
END_DATA_BLOCK

DATA_BLOCK "FV_Regul_2_DB"   // DB21
{ S7_Optimized_Access := 'FALSE' }
VERSION : 0.1
// stored: InstanceOfName Valve(regul)
"Valve(regul)"
BEGIN
END_DATA_BLOCK

DATA_BLOCK "FV_Regul_3_DB"   // DB22
{ S7_Optimized_Access := 'FALSE' }
VERSION : 0.1
// stored: InstanceOfName Valve(regul)
"Valve(regul)"
BEGIN
END_DATA_BLOCK

DATA_BLOCK "FV_Regul_4_DB"   // DB23
{ S7_Optimized_Access := 'FALSE' }
VERSION : 0.1
// stored: InstanceOfName Valve(regul)
"Valve(regul)"
BEGIN
END_DATA_BLOCK

DATA_BLOCK "FV_Regul_5_DB"   // DB37
{ S7_Optimized_Access := 'FALSE' }
VERSION : 0.1
// stored: InstanceOfName Valve(regul)
"Valve(regul)"
BEGIN
END_DATA_BLOCK

// folder: Конвейера/DB

DATA_BLOCK "Конвейер_1_DB"   // DB78
{ S7_Optimized_Access := 'FALSE' }
VERSION : 0.1
// stored: InstanceOfName Pump
"Pump"
BEGIN
END_DATA_BLOCK

DATA_BLOCK "Конвейер_2_DB"   // DB79
{ S7_Optimized_Access := 'FALSE' }
VERSION : 0.1
// stored: InstanceOfName Pump
"Pump"
BEGIN
END_DATA_BLOCK

DATA_BLOCK "Конвейер_3_DB"   // DB80
{ S7_Optimized_Access := 'FALSE' }
VERSION : 0.1
// stored: InstanceOfName Pump
"Pump"
BEGIN
END_DATA_BLOCK

// folder: Насосы/DB

DATA_BLOCK "Pump_6_DB"   // DB5
{ S7_Optimized_Access := 'FALSE' }
VERSION : 0.1
// stored: InstanceOfName Pump
"Pump"
BEGIN
END_DATA_BLOCK

DATA_BLOCK "Pump_7_DB"   // DB7
{ S7_Optimized_Access := 'FALSE' }
VERSION : 0.1
// stored: InstanceOfName Pump
"Pump"
BEGIN
END_DATA_BLOCK

DATA_BLOCK "Pump_1_DB"   // DB25
{ S7_Optimized_Access := 'FALSE' }
VERSION : 0.1
// stored: InstanceOfName Pump
"Pump"
BEGIN
END_DATA_BLOCK

DATA_BLOCK "Pump_2_DB"   // DB26
{ S7_Optimized_Access := 'FALSE' }
VERSION : 0.1
// stored: InstanceOfName Pump
"Pump"
BEGIN
END_DATA_BLOCK

DATA_BLOCK "Pump_5_DB"   // DB27
{ S7_Optimized_Access := 'FALSE' }
VERSION : 0.1
// stored: InstanceOfName Pump
"Pump"
BEGIN
END_DATA_BLOCK

DATA_BLOCK "Pump_4_DB"   // DB28
{ S7_Optimized_Access := 'FALSE' }
VERSION : 0.1
// stored: InstanceOfName Pump
"Pump"
BEGIN
END_DATA_BLOCK

DATA_BLOCK "Pump_3_DB"   // DB29
{ S7_Optimized_Access := 'FALSE' }
VERSION : 0.1
// stored: InstanceOfName Pump
"Pump"
BEGIN
END_DATA_BLOCK

// folder: (top level)

FUNCTION_BLOCK "Pump"   // FB1, SCL
{ S7_Optimized_Access := 'FALSE' }
VERSION : 0.1
   VAR_INPUT
      bManualMode : Bool;   // Выбор ручного режима
      bManualStart : Bool;   // Ручной режим - старт
      bManualStop : Bool;   // Ручной режим - стоп
      rManualSpeed : Real;   // Ручной режим - скорость
      bDryRunn : Bool;   // Защита от сухого хода
      bAutoSTop : Bool;   // Остановка насоса
      bAutoStartPerm : Bool;   // Команда на работоу в авто режиме
      rAutoSpeed : Real;   // Скорость в авто режиме
      bАвтоматы : Bool;   // Готовность привода (автоматы)
      bПускатели : Bool;   // Готовность Пускателя
      bDriveRunning : Bool;   // Привод в работе
      bDriveFault : Bool;   // Привод в ошибке
      rMinSpeed : Real;   // Минимальная скорость
      rMaxSpeed : Real := 100.0;   // Максимальная скорость
      bResetFault : Bool;   // Сброс аварии
   END_VAR
   VAR_OUTPUT
      bRunCmd : Bool;   // Пуск частотника
      iSpeedOut : Int;   // Скорость насоса для аналогового выхода
      "rSpeedHMI(0-100)" : Real;   // Скорость работы (0-100) для HMI
      bPumpRunning : Bool;   // Работа
      bPumpFault : Bool;   // Авария
      iStatus : Int;   // Статус (0 - стоп 1 - работа 2 - авария)
   END_VAR
   VAR
      bFaultLatch : Bool;
      bRunRequest : Bool;
      rSpeedPump : Real;   // Скорость насоса
      TON_NotStartRun : TON_TIME;   // ТАймер ожидания сигнала о запуске
      TON_NotContactRun : TON_TIME;   // ТАймер ожидания с контактора
      TON_DryRun : TON_TIME;   // Таймер сухого хода
   END_VAR
BEGIN
   (*
   // 1. Обработка аварий
   // Обработка ожидания сигнала о работе после старта
   IF #bAutoStartPerm THEN
       ;

   END_IF;
   *)

   // 1 Ручной режим
   IF #bManualMode THEN
       // Ручной режим
       IF #bManualStart AND NOT #bManualStop THEN
           #bRunRequest := TRUE;
       ELSIF #bManualStop THEN // OR NOT #bАвтоматы THEN
           #bRunRequest := FALSE;
       END_IF;
   ELSE
       // Автоматический режим
       // 
       //Обработка аварий
       //
       //Таймер ожидания останова по сухому ходу
       #TON_DryRun(IN := NOT #bDryRunn,
                   PT := t#1s);    //
       //--------------------------------------------------------------------------------------------------------
       IF #bAutoStartPerm AND NOT #bAutoSTop AND #bDryRunn THEN
           #TON_NotStartRun(IN := NOT #bDriveRunning,PT := t#5s);  //Таймер ожидания сигнала подтверждения пуска от частотника
           #TON_NotContactRun(IN := NOT #bПускатели, PT := t#10s);  //Таймер ожидания сигнала подтверждения пуска от пускателя


       ELSE
           #TON_NotStartRun(IN :=FALSE,PT := t#5s);
           #TON_NotContactRun(IN := FALSE,PT := t#5s);
       END_IF;
       #bFaultLatch := #TON_NotStartRun.Q OR #TON_NotContactRun.Q OR (#bDriveFault OR NOT #bАвтоматы) OR (NOT #bResetFault AND #bFaultLatch); //Разкоментировать если нужна будет фиксация АЛАРМА, сброс только по входу РЕСЕТ
       #bPumpFault := #bFaultLatch;

       //Старт--------------------------------
       #bRunRequest := #bAutoStartPerm AND NOT #bPumpFault AND NOT #TON_DryRun.Q;
   END_IF;

   // 3. Задание скорости
   IF #bManualMode THEN
       #"rSpeedHMI(0-100)" := LIMIT(MN := #rMinSpeed, IN := #rManualSpeed, MX := #rMaxSpeed);
   ELSE
       #"rSpeedHMI(0-100)" := LIMIT(MN := #rMinSpeed, IN := #rAutoSpeed, MX := #rMaxSpeed);
   END_IF;

   // Преобразование значения от 0-100 до 0-27648 для аналогового выхода
   #iSpeedOut := REAL_TO_INT((#"rSpeedHMI(0-100)"/ 100.0) * 27648.0);

   // 4. Выходные команды и статусы
   // Команды старт
   #bRunCmd := #bRunRequest;

   //Выход статуса для HMI
   #bPumpRunning := #bDriveRunning AND #bRunCmd AND NOT #bAutoSTop OR (#bManualStart AND #bManualMode);



   // 5. Числовой статус (для HMI/SCADA)
   IF #bFaultLatch THEN
       #iStatus := 2; // Авария
   ELSIF #bPumpRunning THEN
       #iStatus := 1; // Работа
   ELSE
       #iStatus := 0; // Стоп
   END_IF;

   IF #bAutoSTop AND NOT #bManualMode THEN
       #bRunCmd := FALSE;
   END_IF;
END_FUNCTION_BLOCK

FUNCTION_BLOCK "FB_GlobalStateManager"   // FB2, SCL
{ S7_Optimized_Access := 'FALSE' }
VERSION : 0.1
   VAR_INPUT
      bStartCmd : Bool;   // Команда на старт от HMI
      bConfirmStart : Bool;   // Подтверждение оператора
      bResetFault : Bool;   // Сброс ошибки
      bAllSetpointsReached : Bool;   // // Все температуры достигли уставок
      bNoFaults : Bool;   // Нет аварий
      tStartTimeout : Time := T#30m;   // Время за которое пастер выходит на режим
      tReadyDelay : Time := t#10s;   // Время ожидания при выходе на режим до готовности
   END_VAR
   VAR_OUTPUT
      eState : Int;   // Текущее состояние
      bConveyorEnable : Bool;   // Разрешение на работу конвейера
      bSystemReady : Bool;   // Готовность системы
      bSystemFault : Bool;   // Состояние Fault
      sStatusText : WString;   // Текст для HMI
   END_VAR
   VAR
      tonStartTimeout : TON_TIME;   // Таймер выхода на режим
      tonReadyDelay : TON_TIME;   // Таймер готовности
   END_VAR
   VAR CONSTANT
      cSTATE_IDLE : Int;
      cSTATE_CHECK : Int := 10;
      cSTATE_STARTING : Int := 20;
      cSTATE_READY_DELAY : Int := 30;
      cSTATE_READY : Int := 40;
      cSTATE_FAULT : Int := 99;
      sText1 : String := 'Waiting';
   END_VAR
BEGIN
   // Сброс таймеров при неактивных состояниях (по требованию 1)
   IF #eState <> #cSTATE_STARTING THEN
       #tonStartTimeout(IN := FALSE,
                        PT := #tStartTimeout);
   END_IF;

   IF #eState <> #cSTATE_READY_DELAY THEN
       #tonReadyDelay(IN := FALSE,
                      PT := #tReadyDelay);
   END_IF;

   // Глобальная проверка аварии (по требованию 4)
   IF NOT #bNoFaults AND #eState <> #cSTATE_FAULT THEN
       #eState := #cSTATE_FAULT;
       #bSystemFault := TRUE;
       #bConveyorEnable := FALSE; // Принудительный останов (по требованию 2)
   ELSIF NOT #bStartCmd THEN
       #eState := #cSTATE_IDLE;
   END_IF;


   REGION Основная логика

       // Основной CASE
       CASE #eState OF
           #cSTATE_IDLE:
               #bConveyorEnable := FALSE;
               IF #bStartCmd AND #bNoFaults THEN // Запрет старта при аварии
                   #eState := #cSTATE_CHECK;
               END_IF;

           #cSTATE_CHECK:
               // Проверка уже в глобальном условии, дублирование не нужно
               #eState := #cSTATE_STARTING;

           #cSTATE_STARTING:
               IF #bAllSetpointsReached THEN
                   #eState := #cSTATE_READY_DELAY;
               ELSIF #tonStartTimeout.Q THEN
                   #eState := #cSTATE_FAULT;
               END_IF;

           #cSTATE_READY_DELAY:
               IF #tonReadyDelay.Q THEN
                   #eState := #cSTATE_READY;
               END_IF;

           #cSTATE_READY:
               #bSystemReady := TRUE;
               IF #bConfirmStart THEN
                   #bConveyorEnable := TRUE;
               END_IF;

           #cSTATE_FAULT:
               #bSystemFault := TRUE;
               #bConveyorEnable := FALSE; // Гарантированный останов
               IF #bResetFault AND #bNoFaults THEN
                   #eState := #cSTATE_IDLE;
                   #bSystemFault := FALSE;
               END_IF;

           ELSE
               #eState := #cSTATE_IDLE;
       END_CASE;

   END_REGION


   // Обновление таймеров (после логики состояний!)
   #tonStartTimeout(IN := (#eState = #cSTATE_STARTING) AND NOT #bAllSetpointsReached,
                    PT := #tStartTimeout);
   #tonReadyDelay(IN := (#eState = #cSTATE_READY_DELAY),
                  PT := #tReadyDelay);
END_FUNCTION_BLOCK

FUNCTION_BLOCK "Valve(c/o)"   // FB3, SCL
{ S7_Optimized_Access := 'FALSE' }
VERSION : 0.1
   VAR_INPUT
      bAuto_OpenCmd : Bool;   // Команда открыть (автомат)
      bManualMode : Bool;   // Ручной режим (TRUE)
      bManualOpen : Bool;   // Команда открыть в ручном режиме
      bFeedbackOpen : Bool;   // Обратная связь "Открыт"
      tMaxTime : Time;   // Время на открытие
      bResetAlarm : Bool;   // Сброс аварии
      bHaveFeedback : Bool;   // Есть ли обратная связь (0 - нет, 1 есть)
   END_VAR
   VAR_OUTPUT
      bValveOpen : Bool;   // Управляющий выход
      iValveState : Int;   // 0 = Закрыт, 1 = Открыт, 2 = Авария
      bValveFault : Bool;   // Авария
   END_VAR
   VAR
      tiOpenTimer : TON_TIME;   // Таймер на открытие
      bWaitingOpen : Bool;   // Флаг ожидания открытия
      bEnableTimer : Bool;   // Флаг активации таймера
   END_VAR
BEGIN

   // Обновление таймера — всегда в одном месте, вне условий
   #tiOpenTimer(
                IN := #bEnableTimer,
                PT := #tMaxTime
   );

   // Сброс
   IF #bResetAlarm THEN
       #bValveFault := FALSE;
       #bWaitingOpen := FALSE;
       #bEnableTimer := FALSE;
   END_IF;

   // === Режим: РУЧНОЙ ===
   IF #bManualMode THEN
       #bValveOpen := #bManualOpen;
       #bValveFault := FALSE;          // Аварии в ручном режиме не учитываются
       #bEnableTimer := FALSE;
       #bWaitingOpen := FALSE;

       // === Режим: АВТО ===
   ELSE

           // Управление выходом с учетом аварии, с контролем обратной связи
        IF #bAuto_OpenCmd AND NOT #bValveFault THEN
                   #bValveOpen := TRUE;
        ELSE
                   #bValveOpen := FALSE;
               END_IF;

               //  Проверяем, есть ли контроль обратной связи
        IF #bHaveFeedback THEN
            // Контроль открытия
            IF #bAuto_OpenCmd AND NOT #bFeedbackOpen AND NOT #bValveFault THEN
                #bEnableTimer := TRUE;
                #bWaitingOpen := TRUE;
            ELSE
                #bEnableTimer := FALSE;
                ;
                IF #bFeedbackOpen THEN
                    #bWaitingOpen := FALSE;
                END_IF;
            END_IF;
        END_IF;


           // Авария
           IF #tiOpenTimer.Q AND #bWaitingOpen THEN
               #bValveFault := TRUE;
               #bWaitingOpen := FALSE;
           END_IF;

   END_IF;


   // Состояние клапана
   IF #bValveFault THEN
       #iValveState := 2;       // Авария
   ELSIF #bHaveFeedback AND #bFeedbackOpen  THEN
       #iValveState := 1;       // Открыт
   ELSIF NOT #bHaveFeedback AND (NOT #bManualMode AND #bAuto_OpenCmd) OR (#bManualOpen AND #bManualMode) THEN
       #iValveState := 1;       // Открыт 
   ELSE
       #iValveState := 0;       // Закрыт
   END_IF;
END_FUNCTION_BLOCK

FUNCTION_BLOCK "Valve(regul)"   // FB4, SCL
{ S7_Optimized_Access := 'FALSE' }
VERSION : 0.1
   VAR_INPUT
      bManualMode : Bool;   // TRUE = ручной режим, FALSE = автоматический режим
      rAutoSetpoint : Real;   // Уставка открытия клапана в % (0.0–100.0) в автомате
      "bAutoOpen/Close" : Bool;   // Выход Do в автоматическом режиме
      rManualSetpoint : Real;   // Уставка открытия клапана в % (0.0–100.0) в ручном режиме
      "bManualOpen/Close" : Bool;   // Управление выходом открыть/закрыть
   END_VAR
   VAR_OUTPUT
      iAnalogOutput : Int;   // Значение для аналогового выхода (0–27648)
      rValvePosPercent : Real;   // Текущее % открытия клапана для HMI
      bStatusValveOpen : Int;   // Статус сигнал "клапан открыт" (TRUE, если >0%)
      "bOut_Open/Close" : Bool;   // выход для открытия клапана
   END_VAR
   VAR
      rSetpointPercent : Real;   // Расчётная уставка % открытия в текущем режиме
   END_VAR
BEGIN
       // Выбор уставки в зависимости от режима
       IF #bManualMode THEN
           #rSetpointPercent := #rManualSetpoint;
           #"bOut_Open/Close" := #"bManualOpen/Close";
       ELSE
           #rSetpointPercent := #rAutoSetpoint;
           #"bOut_Open/Close" := #"bAutoOpen/Close";
       END_IF;

       // Ограничение % от 0.0 до 100.0
       IF #rSetpointPercent < 0.0 THEN
           #rSetpointPercent := 0.0;
       ELSIF #rSetpointPercent > 100.0 THEN
           #rSetpointPercent := 100.0;
       END_IF;

       // Перевод % в значение для аналогового выхода
       #iAnalogOutput := REAL_TO_INT((#rSetpointPercent / 100.0) * 27648.0);

           // Вывод значения для HMI
       #rValvePosPercent := #rSetpointPercent;

       // Статус клапана для Панели HMI
       IF #rSetpointPercent > 0.0 AND #"bOut_Open/Close" THEN
           #bStatusValveOpen := 1;
       ELSE
           #bStatusValveOpen := 0;
       END_IF;
       ;
END_FUNCTION_BLOCK

FUNCTION_BLOCK "FB_Управление конвейером"   // FB5, SCL
{ S7_Optimized_Access := 'FALSE' }
VERSION : 0.1
   VAR_INPUT
      bEnable : Bool;   // Общий флаг работы системы
      bStartCmd : Bool;   // Команда на запуск от HMI, по кнопке из окна подтверждения
      bAllZonesInSetpoint : Bool;   // Все зоны достигли уставок
      bGlobalFault : Bool;   // Авария по системе
      bZoneHasPriority : Bool;   // У зоны с отклонением есть приоритет
      dwDeltaTempDelayMin : DWord;   // Задержка (мин), прежде чем остановить конвейер при отклонении
      dwResumeDelayMin : DInt;   // Время возврата после нормализации
   END_VAR
   VAR_OUTPUT
      bConveyorRun : Bool;   // Команда на пуск частотников
      bReadyToStart : Bool;   // Готовность к работе конвейера
      bWaitingConfirm : Bool;   // Ждём подтверждения от оператора, вывод окна на HMI
      bPaused : Bool;   // Конвейер остановлен по отклонению
   END_VAR
   VAR
      bStarted : Bool;   // Внутреннее состояние — процесс стартовал
      tiPauseTimer : TON_TIME;   // Таймер задержки перед остановкой
      tiResumeTimer : TON_TIME;   // Таймер ожидания перед возобновлением
      aZoneS_Status : Array[1..5] of "ZoneStatus";   // Массив для сбора состояния зон
      i : Int;
   END_VAR
   // tiPauseTimer.PT := T#1s;
   // tiResumeTimer.PT := T#1s;
BEGIN

   // Проверка на наличие флага обей работы системы
   IF NOT #bEnable THEN
       #bReadyToStart := FALSE;
       #bWaitingConfirm := FALSE;
       #bConveyorRun := FALSE;
       #bPaused := FALSE;
       #tiPauseTimer.IN := FALSE;
       #tiResumeTimer.IN := FALSE;
       RETURN;
   END_IF;



   // Условия готовности к запуску
   IF NOT #bStarted AND NOT #bGlobalFault AND #bAllZonesInSetpoint THEN
       #bReadyToStart := TRUE;

           // Команда на старт — вручную подтверждена
           IF NOT #bStartCmd THEN
               #bWaitingConfirm := TRUE;
           END_IF;

   ELSE
       #bReadyToStart := FALSE;
       #bWaitingConfirm := FALSE;
   END_IF;



   IF #bStartCmd AND #bReadyToStart THEN
       #bStarted := TRUE;
       #bWaitingConfirm := FALSE;
   END_IF;

   // После старта разрешаем работу, если нет аварий и температур в норме
   IF #bStarted AND NOT #bGlobalFault THEN

       IF NOT #bAllZonesInSetpoint THEN
           IF #bZoneHasPriority THEN
               // Включаем таймер паузы, задержка перед остановкой
               #tiPauseTimer(IN := TRUE,
                             PT := (#dwDeltaTempDelayMin * 60000)) //В минутах
               ;
           ELSE
               #tiPauseTimer(IN := FALSE,PT := t#0s);
           END_IF;

           // Переход в паузу
           IF #tiPauseTimer.Q THEN
               #bPaused := TRUE;
               #bConveyorRun := FALSE;
               #tiResumeTimer(IN := FALSE, PT := t#0s); // Сброс таймера возобновления

           END_IF;

       ELSE
           // Температуры вернулись в норму — запускаем таймер на возврат
           IF #bPaused THEN
               #tiResumeTimer(IN := TRUE,
                              PT := (#dwResumeDelayMin * 60000)) // в минутах
               ;
               // Возвращаемся к работе
               IF #tiResumeTimer.Q THEN
                   #bPaused := FALSE;
                   #bConveyorRun := TRUE;
                   #tiResumeTimer(IN := FALSE, PT := t#0s); // сброс таймера
               END_IF;
           ELSE
               #bConveyorRun := TRUE;
               #tiPauseTimer(IN := FALSE, PT := t#0s); // сброс
               #tiResumeTimer(IN := FALSE,PT := t#0s);
           END_IF;
       END_IF;
   ELSE
       // Если глобальная авария — всё стоп
       #bConveyorRun := FALSE;
       #bPaused := FALSE;
       #bStarted := FALSE;
       #tiPauseTimer(IN := FALSE, PT := t#0s);
       #tiResumeTimer(IN := FALSE,PT := t#0s);
       #bWaitingConfirm := FALSE;
   END_IF;
END_FUNCTION_BLOCK

FUNCTION_BLOCK "FB_Motor_Conveyor"   // FB6, SCL
{ S7_Optimized_Access := 'FALSE' }
VERSION : 0.1
   VAR_INPUT
      bManualMode : Bool;   // Выбор ручного режима
      bManualStart : Bool;   // Ручной режим - старт
      bManualStop : Bool;   // Ручной режим - стоп
      rManualSpeed : Real;   // Ручной режим - скорость
      bAutoStartPerm : Bool;   // Команда на работоу в авто режиме
      rAutoSpeed : Real;   // Скорость в авто режиме
      bDriveReady : Bool;   // Готовность привода (автоматы)
      bDriveRunning : Bool;   // Привод в работе
      bDriveFault : Bool;   // Привод в ошибке
      rMinSpeed : Real;   // Минимальная скорость
      rMaxSpeed : Real;   // Максимальная скорость
      bResetFault : Bool;   // Сброс аварии
   END_VAR
   VAR_OUTPUT
      bRunCmd : Bool;   // Пуск частотника
      "rSpeedHMI(0-100)" : Real;   // Скорость работы (0-100) для HMI
      iSpeedOut : Int;   // Скорость насоса для аналогового выхода
      bPumpRunning : Bool;   // Работа
      bPumpFault : Bool;   // Авария
      iStatus : Int;   // Статус (0 - стоп 1 - работа 2 - авария)
   END_VAR
   VAR
      bFaultLatch : Bool;
      bRunRequest : Bool;
      rSpeedPump : Real;   // Скорость насоса
   END_VAR
BEGIN
   // 1. Обработка аварий
   #bFaultLatch := (#bDriveFault OR #bFaultLatch) AND NOT #bResetFault;
   #bPumpFault := #bFaultLatch;

   // 2. Формирование команды "Пуск"
   IF #bManualMode THEN
       // Ручной режим
       IF #bManualStart AND NOT #bManualStop THEN
           #bRunRequest := TRUE;
       ELSIF #bManualStop OR NOT #bDriveReady THEN
           #bRunRequest := FALSE;
       END_IF;
   ELSE
       // Автоматический режим
       #bRunRequest := #bAutoStartPerm AND NOT #bDriveFault;
   END_IF;

   // 3. Задание скорости
   IF #bManualMode THEN
       #"rSpeedHMI(0-100)" := LIMIT(MN := #rMinSpeed, IN := #rManualSpeed, MX := #rMaxSpeed);
   ELSE
       #"rSpeedHMI(0-100)" := LIMIT(MN := #rMinSpeed, IN := #rAutoSpeed, MX := #rMaxSpeed);
   END_IF;

   // Преобразование значения от 0-100 до 0-27648 для аналогового выхода
   #iSpeedOut := REAL_TO_INT((#"rSpeedHMI(0-100)"/ 100.0) * 27648.0);

   // 4. Выходные команды и статусы
   #bRunCmd := #bRunRequest AND NOT #bFaultLatch AND #bDriveReady;
   #bPumpRunning := #bDriveRunning AND #bRunCmd;

   // 5. Числовой статус (для HMI/SCADA)
   IF #bFaultLatch THEN
       #iStatus := 2; // Авария
   ELSIF #bPumpRunning THEN
       #iStatus := 1; // Работа
   ELSE
       #iStatus := 0; // Стоп
   END_IF;
END_FUNCTION_BLOCK

FUNCTION_BLOCK "FB_Аварии"   // FB7, SCL
{ S7_Optimized_Access := 'FALSE' }
VERSION : 0.1
   VAR_INPUT
      Rtrig_Reset : Bool;
   END_VAR
   VAR_OUTPUT
      ALARM_Active : Bool;   // Флаг активной аварии
   END_VAR
   VAR
      LatchedEmergency : Bool;   // Зафиксированная аварийная ситуация
      bAlarmAvtomats : Bool;   // Авария автоматов
      bAlarmAI : Bool;   // Авария аналоговых датчиков
      bAlarmPumps : Bool;   // Авария насосов
      bAlarmConveyors : Bool;   // Авария Конвейеров
      bAlarmFVs : Bool;   // Авария клапанов
      bAlarmDI_all : Bool;   // Авария по дискретным входам "общая"
      bAlarmLowLevel : Bool;   // Авария по низкому уровню емкостей
      mReset : Bool;
      TON_LowLevel : TON_TIME;   // Таймер для аварийного уровня емкостей
      bResetaALARM : Bool;   // Сброс аварии (кнопка на панели/системе)
   END_VAR
   VAR_TEMP
      nAi : Int;
      nPump : Int;
      nConv : Int;
      nFV : Int;
      nAvtomat : Int;
      numPump : Int;
   END_VAR
BEGIN
   REGION Предварительное отрицание
       // Сброс в 0 при отсутсвии аварий для цикла и массивов
       #bAlarmAvtomats := FALSE;
       #bAlarmAI := FALSE;
       #bAlarmPumps := FALSE;
       #bAlarmConveyors := FALSE;
       #bAlarmFVs := FALSE;


   END_REGION



   //Авария автоматические выключатели
   //--------------------------
   //
   "Alarms".Avtomat_Off[1].ALARM := NOT "Conveyor".Conveyor_1.bIn_AutomatState;
   "Alarms".Avtomat_Off[2].ALARM := NOT "Conveyor".Conveyor_2.bIn_AutomatState;
   "Alarms".Avtomat_Off[3].ALARM := NOT "Conveyor".Conveyor_3.bIn_AutomatState;
   "Alarms".Avtomat_Off[4].ALARM  :=  NOT "Pumps".Pump_1.bIn_AutomatState;
   "Alarms".Avtomat_Off[5].ALARM  :=  NOT "Pumps".Pump_2.bIn_AutomatState;
   "Alarms".Avtomat_Off[6].ALARM  :=  NOT "Pumps".Pump_3.bIn_AutomatState;
   "Alarms".Avtomat_Off[7].ALARM  :=  NOT "Pumps".Pump_4.bIn_AutomatState;
   "Alarms".Avtomat_Off[8].ALARM  :=  NOT "Pumps".Pump_5.bIn_AutomatState;
   "Alarms".Avtomat_Off[9].ALARM  :=  NOT "Pumps".Pump_6.bIn_AutomatState;
   "Alarms".Avtomat_Off[10].ALARM  :=  NOT "Pumps".Pump_7.bIn_AutomatState;
   "Alarms".Avtomat_Off[11].ALARM  :=  NOT "Vent".Vent_1.bIn_AutomatState;


   FOR #nAvtomat := 1 TO 11 DO
       IF "Alarms".Avtomat_Off[#nAvtomat].ALARM THEN
           #bAlarmAvtomats := TRUE;
       END_IF;
   END_FOR;

   //Авария аналоговых входов
   //--------------------------
   FOR #nAi := 1 TO 7 DO
       IF "Alarms".Ai_Alarm[#nAi].ALARM THEN
           #bAlarmAI := TRUE;
       END_IF;
   END_FOR;

   //Авария НАСОСОВ
   //--------------------------

   FOR #nPump := 1 TO 7 DO
       IF "Alarms".Pump_Alarm[#nPump].ALARM THEN
           #bAlarmPumps := TRUE;
           #numPump := #nPump;

       END_IF;
   END_FOR;

   //Авария КОНВЕЙЕРОВ
   //--------------------------

   FOR #nConv := 1 TO 4 DO
       IF "Alarms".Conveyor_Alarm[#nConv].ALARM THEN
           #bAlarmConveyors := TRUE;
       END_IF;
   END_FOR;

   //Авария Клапанов
   //--------------------------

   FOR #nFV := 1 TO 7 DO
       IF "Alarms".FV_Alarm[#nFV].ALARM THEN
           #bAlarmFVs := TRUE;
       END_IF;
   END_FOR;

   //Авария под давлению
   //--------------------------
   "AlarmPress" := "Control_Press_DB".PressWater.bAlarm_Press OR "Control_Press_DB".PressSteam.bAlarm_Press OR "Control_Press_DB".PressGlikol.bAlarm_Press;

   //Авария по нижним датчикам уровня емкостей
   //

   //#bAlarmLowLevel := NOT "My_VarS".b_Woter_LowLevel_T1;

   //Авария по входам DI
   //---------------------------

   #bAlarmDI_all :="Alarms"."xE-Stop_1" OR
                   "Alarms"."xE-Stop_2" OR
                   "Alarms"."xE-Stop_3" OR
                   "Alarms".xVoltRele OR
                   "Alarms".xSensorConveyorZator_1 OR
                  // "Alarms".xSensorConveyorZator_2 OR
                   "Alarms".xLongPauseConv OR
                   "Alarms".xLongWaitZoneOk;

   //Обработка всех аварий с выводом сигнала наличия АВАРИЯ
   //----------------------------------------------------------------
                   IF #bAlarmAvtomats OR
                       #bAlarmAI OR
                       #bAlarmPumps OR
                       #bAlarmConveyors OR
                       #bAlarmFVs OR
                       #bAlarmDI_all OR
                       #bAlarmLowLevel
                   THEN

                       #ALARM_Active := TRUE;
                   END_IF;
     (*                     
   //Отлавливаем фронт Ресета....................................

   #bResetaALARM := #Rtrig_Reset AND NOT #mReset;
   #mReset := #Rtrig_Reset;
   *)

    //Если нужен жесткий сбро, игнорирует все аварии                      
   #bResetaALARM := #Rtrig_Reset;

   //-------------------------------------------------------------                       
                          // Сброс аварии
   IF #bResetaALARM THEN
       #ALARM_Active := FALSE;
   END_IF;
END_FUNCTION_BLOCK

FUNCTION_BLOCK "FB_Zone_Control"   // FB8, SCL
{ S7_Optimized_Access := 'FALSE' }
VERSION : 0.1
   VAR_INPUT
      bNewStart : Bool;   // Обнаружение нового старта, уставка без дельты
      rTempActual : Real;   // Температура с датчика
      rTempSetpoint : Real;   // Уставка температуры
      rDeltaDown : Real;   // Верхнее Допустимое отклонение от уставки
      rDeltaUp : Real;   // Верхнее Допустимое отклонение от уставки
      bPriority : Bool;   // Приоритет управления конвейером (1 - стоп конвейер)
   END_VAR
   VAR_OUTPUT
      ZoneStatusOut : "ZoneStatus";
      bInSetpoint : Bool;
      bOutOfRange : Bool;
      bHasPriority : Bool;
   END_VAR
   VAR
      R_Trig_Start : "R_trig";
      "#bNewStartCLic" : Bool;
      bSetpointReachedOnce : Bool;
   END_VAR
BEGIN
   // --- Сброс флага при необходимости ---
   // 
       //----Отслеживание нажания старта, по верхнему фронту-----
   #R_Trig_Start("In":= #bNewStart,Q => #"#bNewStartCLic");

   IF #"#bNewStartCLic" THEN
       #bSetpointReachedOnce := FALSE;
   END_IF;

   // --- Фиксация первого достижения уставки (точно или ±0.1) ---
   IF NOT #bSetpointReachedOnce AND ABS(#rTempActual - #rTempSetpoint) <= 1 THEN
       #bSetpointReachedOnce := TRUE;
   END_IF;

   // --- Расчёт попадания в уставку с учетом асимметричной дельты ---
   IF #bSetpointReachedOnce THEN
       #ZoneStatusOut.bInSetpoint := (#rTempActual >= (#rTempSetpoint - #rDeltaDown)) AND
                                       (#rTempActual <= (#rTempSetpoint + #rDeltaUp));
   ELSE
       // До первого достижения — строгое приближение (или узкая дельта)
       #ZoneStatusOut.bInSetpoint := ABS(#rTempActual - #rTempSetpoint) <= 1;
   END_IF;

   //Контроль зоны выхода из уставок значительно, греем снова до уставки до разрешения на старт

   IF (#rTempActual < (#rTempSetpoint - #rDeltaDown)) OR
       (#rTempActual > (#rTempSetpoint + #rDeltaUp)) THEN
       #bSetpointReachedOnce := FALSE;
   END_IF;


   // --- Остальные сигналы ---
   #ZoneStatusOut.bOutOfRange := NOT #ZoneStatusOut.bInSetpoint;
   #ZoneStatusOut.bHasPriority := #bPriority;

   // Зеркалируем, если нужно
   #bInSetpoint := #ZoneStatusOut.bInSetpoint;
   #bOutOfRange := #ZoneStatusOut.bOutOfRange;
   #bHasPriority := #ZoneStatusOut.bHasPriority;
END_FUNCTION_BLOCK

FUNCTION_BLOCK "FB_check_For_Start"   // FB9, SCL
{ S7_Optimized_Access := 'FALSE' }
VERSION : 0.1
   VAR_INPUT
      xHMI_Start : Bool;   // кнопка старта с HMI
      xEmergency_Stop : Bool;   // аварийный стоп
      xSystem_Ready : Bool;   // Готовность всех систем
      xStopHMI : Bool;   // Кнопка СТОП на HMI
   END_VAR
   VAR_OUTPUT
      xStart_Allowed : Bool;   // Разрешение на РАБОТУ
      xStart : Bool;   // Работа пастеризатора
   END_VAR
   VAR
      "m" : Bool;   // memory
   END_VAR
BEGIN

   //Проверка на разрешение работы.
   //
   IF NOT #xEmergency_Stop AND #xSystem_Ready THEN
       #xStart_Allowed := TRUE;
   ELSE
       #xStart_Allowed := FALSE;
   END_IF;

   #xStart := (#xStart OR #xHMI_Start) AND NOT (#xEmergency_Stop OR #xStopHMI);
END_FUNCTION_BLOCK

FUNCTION_BLOCK "FB_Stiril_CheckZoneStatus"   // FB10, SCL
{ S7_Optimized_Access := 'FALSE' }
VERSION : 0.1
   VAR_OUTPUT
      bAllZones_Redy : Bool;   // Выход состояния всех зон ОК
      bPriority_Stop : Bool;   // Выход 1 - если есть метка остановки конвейера
      iZonesNumberFail : Int;   // ВЫход с Номером зоны
   END_VAR
   VAR
      aZoneS_Status : Array[1..7] of "ZoneStatus";   // Массив с данными по всем зонам
      i : Int;
      AllZone_Ok : Bool;   // Состояние всех зон ОК
      HaveStopPriority : Bool;   // В зоне есть метка для остановки конвейера
      iNumber : Int;   // Номер зоны, где отклонение температуры
   END_VAR
BEGIN

   //Что бы не контролировал готовность зоны 4 ее не надо контролировать
   //"ЗОНЫ_Параметры".Zone_4.bOUT_ZoneStatus.bInSetpoint := TRUE;
   //-------------------------------------------------------------------------------------------//
   //
           // ----Сбор данных по всем зонам в массив для обработки-----
           #aZoneS_Status[1] := "Зоны_Стерилизации_Парам"."Steril_Zona-1".bOUT_ZoneStatus;
           #aZoneS_Status[2] := "Зоны_Стерилизации_Парам"."Steril_Zona-2".bOUT_ZoneStatus;
           #aZoneS_Status[3] := "Зоны_Стерилизации_Парам"."Steril_Zona-3".bOUT_ZoneStatus;
           #aZoneS_Status[4] := "Зоны_Стерилизации_Парам"."Steril_Zona-4".bOUT_ZoneStatus;
           #aZoneS_Status[5] := "Зоны_Стерилизации_Парам"."Steril_Zona-5".bOUT_ZoneStatus;
           #aZoneS_Status[6] := "Зоны_Стерилизации_Парам"."Steril_Zona-6".bOUT_ZoneStatus;
           #aZoneS_Status[7] := "Зоны_Стерилизации_Парам"."Steril_Zona-7".bOUT_ZoneStatus;


           //Сброс маркеров по умолчанию----
   #AllZone_Ok := TRUE;    
   #HaveStopPriority := FALSE;
   #iNumber := 0;
              // ----Цикл для перебора всех зон значение выставить по количеству зон----
   FOR #i := 1 TO 7 DO
       IF NOT #aZoneS_Status[#i].bInSetpoint THEN
           #AllZone_Ok := FALSE;
           #iNumber := #i;
           IF #aZoneS_Status[#i].bHasPriority THEN
               #HaveStopPriority := TRUE;
           END_IF;
       END_IF;
   END_FOR;

   /// Присвоение переменных к выходам
   #bAllZones_Redy := #AllZone_Ok;
   #bPriority_Stop := #HaveStopPriority;
   #iZonesNumberFail := #iNumber;
END_FUNCTION_BLOCK

FUNCTION_BLOCK "FB_ПЕ_Control"   // FB11, SCL
{ S7_Optimized_Access := 'TRUE' }
VERSION : 0.1
   VAR_INPUT
      bRunRequest : Bool;   // Запрос на работу
      rSpeedPercent : Real;   // Заданная скорость от оператора (0…100%)
      rPESetpoint : Real;   // Заданное количество ПЕ
      rConveyorLength : Real := 8.3;   // Длина зоны выдержки, м
      rVmax : Real := 0.0085;   // Макс скорость м/мин
      rZParam : Real := 1.393;   // Коэффициент z (1.393 обычно)
      rTref : Real := 60.0;   // Базовая температура (обычно 60°C)
      rTmin : Real;   // Мин допустимая температура
      rTmax : Real := 75.0;   // Макс допустимая температура
      bManualMode : Bool;   // Режим "ручной расчёт температуры"
      rManualTemp : Real;   // Температура в ручном режиме
      tStopTolerance : Time;   // Допустимое время простоя
   END_VAR
   VAR_OUTPUT
      rTempSetpoint : Real;   // Уставка температуры
      rHoldTime : Real;   // Время выдержки в мин
      rConveyorSpeed : Real;   // Скорость конвейера (м/мин)
      rPENeededPerMin : Real;   // Требуемое ПЕ в минуту
      bTempValid : Bool;   // Температура в пределах допустимого
      bAlarmTempHigh : Bool;   // Температура превышает максимум
      bAlarmTempLow : Bool;   // Температура ниже минимума
      bStoppedTooLong : Bool;   // Превышено время простоя
      bAlarmTempOverride : Bool;   // Принудительная уставка из-за аварии
   END_VAR
   VAR RETAIN
      rSpeedRatio : Real;   // Отношение скорости
      rLogArg : Real;   // Аргумент логарифма
   END_VAR
   VAR
      TON_StopDelay : TON_TIME;   // Таймер задержки останова
   END_VAR
BEGIN
   // Блок управления уставкой температуры по ПЕ и скорости
   // Сначала сброс в случае остановки
   IF NOT #bRunRequest THEN
       //#rTempSetpoint := 0.0;
       #rHoldTime := 0.0;
       #rConveyorSpeed := 0.000;
       #bTempValid := TRUE;
       #bAlarmTempHigh:= FALSE;
       #bAlarmTempLow := FALSE;
       #bAlarmTempOverride := FALSE;
       #bStoppedTooLong := FALSE;
       #TON_StopDelay(IN := FALSE, PT := t#0s);
       //RETURN;
   END_IF;


   // Преобразуем % скорости в отношение
   #rSpeedRatio := #rSpeedPercent / 100.0;

   // Расчёт фактической скорости (м/с)
   #rConveyorSpeed := #rVmax * #rSpeedRatio;

   // Время нахождения бутылки в зоне (мин)
   IF #rConveyorSpeed > 0.0 THEN
       #rHoldTime := #rConveyorLength / #rConveyorSpeed; // В мин
   ELSE
       #rHoldTime := 0.0;
   END_IF;


   IF #bManualMode THEN
       // Ручной режим — берём температуру с панели
       #rTempSetpoint := #rManualTemp;
   ELSE
       // Расчёт температуры по ПЕ
       IF #rHoldTime > 0.0 AND #rPESetpoint > 0.0 THEN
           #rPENeededPerMin := #rPESetpoint / #rHoldTime;
           #rTempSetpoint := #rTref + (LN(#rPENeededPerMin) / LN(#rZParam));


           (*
           #rLogArg := LN(#rPENeededPerMin) / LN(10.0);
           #rTempSetpoint := #rTref + #rLogArg / #rZParam;
           *)
       ELSE
           #rTempSetpoint := #rTref; // по умолчанию
       END_IF;
   END_IF;

   // Проверка пределов
   #bTempValid := TRUE;
   #bAlarmTempHigh := FALSE;
   #bAlarmTempLow := FALSE;


   IF #rTempSetpoint > #rTmax THEN
       #rTempSetpoint := #rTmax;
       #bTempValid := FALSE;
       #bAlarmTempHigh := TRUE;
   ELSIF #rTempSetpoint < #rTmin THEN
       #rTempSetpoint := #rTmin;
       #bTempValid := FALSE;
       #bAlarmTempLow := TRUE;
   END_IF;
END_FUNCTION_BLOCK

FUNCTION_BLOCK "FB_Главный блок конвейера"   // FB12, SCL
{ S7_Optimized_Access := 'TRUE' }
VERSION : 0.1
   VAR_INPUT
      bModePaster : Bool;   // Режим пастеризации
      bModeStiril : Bool;   // Режим сетрилизации
      bAlarmSystem : Bool;   // Общая авария
      bResAlarm : Bool;   // Сброс аварий
      bStartCMD : Bool;   // Подтверждение оператором старта
      bAllZone_Ok : Bool;   // Маркер - все зоны ОК
      bHasPauseKonv : Bool;   // Маркер - пауза конвейера
      tiWaitZone : DInt;   // HMI - мин - Время ожидания выхода на режим
      tiWaitPause : DInt;   // HMI - мин - Время ожидания возврата с паузы
      tiWaitToGoPause : DInt;   // HMI-сек Время задержки для перехода на паузу
      tiWaitToCameGo : DInt;   // HMI- сек Время задержки для возврата в рабочий режим
   END_VAR
   VAR_OUTPUT
      iStep : Int;   // Шаг конвейера
      bKonveyorRun : Bool;   // Разрешение на работу конвейера
      bAlarmToLongPause : Bool;   // Авария по превышения ожидания выхода с паузы
      bAlarmToLongWaitZone_Ok : Bool;   // Авария по превышения ожидания выхода на режим
      bOpenWindOper : Bool;   // вызов окна оператора
   END_VAR
   VAR
      TON_WaitZones : TON_TIME;   // Таймер ожидания перехода в готовность, или в Аварию
      TON_PauseWait : TON_TIME;   // Таймер ожидания возврата с паузы до перехода в аварию
      TON_WaitToGoPaus : TON_TIME;   // Задержка для перехода в паузу
      TON_WaitToComeGo : TON_TIME;   // Задержка для выхода из паузу
      bAlarm_Timer : Bool;   // общий меркер по авариям внутри конве
   END_VAR
   VAR CONSTANT
      S_STOP : Int;   // Шаги
      S_Start_WaitZones : Int := 10;
      S_ConfirmStart : Int := 20;
      S_Working : Int := 30;
      S_Paused : Int := 40;
      S_Sterilization : Int := 50;
      S_Alarm : Int := 99;
      ConstMin : DInt := 60000;   // Минуты
      ConstS : DInt := 1000;   // Секунды
   END_VAR
BEGIN

   // Проверяем блок на наличие внешних аварий и наличие разрешения на работу
   #bOpenWindOper := FALSE;


   IF #bAlarmSystem OR #bAlarm_Timer THEN
       #iStep := #S_Alarm;
   ELSIF
       NOT #bModePaster AND NOT #bModeStiril AND NOT (#iStep = #S_Alarm) THEN
       #iStep := #S_STOP;
   END_IF;


   CASE #iStep OF
           //...................................................................................................................................................        
       #S_STOP: // ШАГ - СТОП 0
           //....Сбрасываем таймеры.......
           #TON_WaitToGoPaus(IN := FALSE,
                             PT := t#0s);
           #TON_WaitToComeGo(IN := FALSE,
                             PT := t#0s);
           #TON_WaitZones(IN := FALSE,
                          PT := t#0s);
           #TON_PauseWait(IN := FALSE,
                          PT := t#0s);

           #bKonveyorRun := FALSE;


           IF #bModePaster THEN
               #iStep := #S_Start_WaitZones;
           ELSIF #bModeStiril THEN
               #iStep := #S_Sterilization;
           END_IF;

           //...................................................................................................................................................
       #S_Start_WaitZones: // Шаг - Ожидание готовности зон 10
           IF #bAllZone_Ok THEN
               // Если все зоны впорядке сбрасывам таймер ожидания готовности зоны
               #TON_WaitZones(IN := FALSE,
                              PT := #tiWaitZone * #ConstMin);
               #iStep := #S_ConfirmStart;
           ELSE
               #TON_WaitZones(IN := TRUE,
                              PT := #tiWaitZone * #ConstMin);
               IF #TON_WaitZones.Q THEN
                   #bAlarmToLongWaitZone_Ok := TRUE;
                   #iStep := #S_STOP;
               END_IF;
           END_IF;

           //...................................................................................................................................................
       #S_ConfirmStart:    // ШАГ ожидания подтверждения оператора 20
           #bOpenWindOper := #bAllZone_Ok;
           IF #bAllZone_Ok THEN    // Если все зоны готовы то выводим окно оператора и ждем подтверждения
               #bOpenWindOper := TRUE; //Вызов окна оператора
               IF #bStartCMD THEN
                   //#bOpenWindOper := FALSE;
                   #iStep := #S_Working;
               END_IF;
           ELSE
               #iStep := #S_Start_WaitZones;
           END_IF;

           //...................................................................................................................................................            
       #S_Working:         // ШАГ Работа конвейера 30
           IF NOT #bAllZone_Ok THEN
               IF #bHasPauseKonv THEN
                   #TON_WaitToGoPaus(IN := TRUE,
                                     PT := #tiWaitToGoPause * #ConstS);
                   IF #TON_WaitToGoPaus.Q THEN
                       #iStep := #S_Paused;
                   END_IF;
               END_IF;
           ELSE
               #bKonveyorRun := TRUE;

               #TON_WaitToGoPaus(IN := FALSE,
                                 PT := t#0s);
           END_IF;

           //...................................................................................................................................................              
       #S_Paused:          //ШАГ Пауза 40

           #bKonveyorRun := FALSE;

           //Запускаем таймер ожидания предельного времени нахождения в паузе
           #TON_PauseWait(IN := TRUE,
                          PT := #tiWaitPause * #ConstMin);

           // Проверка таймера - если время вышло то АВАРИЯ
           IF #TON_PauseWait.Q THEN
               #bAlarmToLongPause := TRUE;
               #iStep := #S_STOP;
           END_IF;

           // Проверка возврата в рабочий режим - если маркер паузы снят, то возвращаемся в старт
           IF NOT #bHasPauseKonv THEN
               //Сброс таймера Пауза
               #TON_PauseWait(IN := FALSE,
                              PT := t#0s);
               //Старт таймер ожидания возврата к работе
               #TON_WaitToComeGo(IN := TRUE,
                                 PT := #tiWaitToCameGo * #ConstS);

               IF #TON_WaitToComeGo.Q THEN
                   #iStep := #S_Working;
               END_IF;
           ELSE
               #TON_WaitToComeGo(IN := FALSE,
                                 PT := #tiWaitToCameGo * #ConstS);
           END_IF;


           //...................................................................................................................................................              
       #S_Sterilization:          //ШАГ Сттерилизиция

           #bKonveyorRun := FALSE;         //Conveyor - STOP

           //....................................................................................................................................................
           //____________________ Alarm ____________________________

       #S_Alarm:
           #bKonveyorRun := FALSE;
           IF #bResAlarm THEN
               #iStep := #S_STOP;
           END_IF;

   END_CASE;

   // Сброс Аварий
   IF #bResAlarm THEN
       #bAlarmToLongPause := FALSE;
       #bAlarmToLongWaitZone_Ok := FALSE;
   END_IF;
   // Вызов окна подтверждения оператора

   //Флаг АВАРИИ внутренний по таймерам
   #bAlarm_Timer := #bAlarmToLongWaitZone_Ok OR #bAlarmToLongPause;
END_FUNCTION_BLOCK

FUNCTION_BLOCK "FB_Filling_Bac"   // FB17, SCL
{ S7_Optimized_Access := 'TRUE' }
VERSION : 0.1
   VAR_INPUT
      bLevelLow : Bool;   // Датчик нижнего уровня
      bLevelHigh : Bool;   // Датчик верхнего уровня
      bEnable : Bool;   // Разрешение на работу
      bManualMode : Bool;   // Ручной режим
      bManualOpen : Bool;   // Принудительно открыть клапан в ручном режиме
      tDelayOff : Time := T#2s;   // Задержка отключения после высокого уровня
   END_VAR
   VAR_OUTPUT
      bValveOpen : Bool;   // Управление клапаном
   END_VAR
   VAR
      bFilling : Bool;   // Внутренний флаг процесса наполнения
      tonDelayOff : TON_TIME;   // Таймер задержки отключения
      tonDelayOn : TON_TIME;   // Таймер задержки включения
   END_VAR
BEGIN

   // Режим ручного управления
   IF #bManualMode THEN
       #bValveOpen := #bManualOpen;

   ELSE
       // Автоматический режим
       IF NOT #bEnable THEN
           // Если нет разрешения — всё выключено
           #bFilling := FALSE;
           #tonDelayOff(IN := FALSE,PT := t#0s);
           #tonDelayOff(IN := FALSE,PT := t#0s);
           #bValveOpen := FALSE;

       ELSE
           // Основная логика управления
           IF NOT #bLevelHigh THEN
               // Запускаем таймер на включение наполнения
               #tonDelayOn(IN := TRUE,
                           PT := #tDelayOff*1000);

               // Включаем наполнение емкостей
               #bFilling := #tonDelayOn.Q;
           ELSE
               #tonDelayOn(IN := FALSE,
                           PT := #tDelayOff * 1000);
           END_IF;

           IF #bLevelHigh THEN
               // Запускаем таймер задержки отключения в секундах
               #tonDelayOff(IN := TRUE,
                            PT := #tDelayOff*1000);

               // Если задержка прошла — отключаем наполнение
               IF #tonDelayOff.Q THEN
                   #bFilling := FALSE;
               END_IF;
           ELSE
               // Если уровень упал — сбрасываем таймер
               #tonDelayOff(IN := FALSE, PT := t#0s);
           END_IF;

           #bValveOpen := #bFilling;
       END_IF;
   END_IF;
END_FUNCTION_BLOCK

FUNCTION_BLOCK "FB_Press_Controll"   // FB18, SCL
{ S7_Optimized_Access := 'TRUE' }
VERSION : 0.1
   VAR_IN_OUT
      DataPress : "tipePress";
   END_VAR
   VAR
      TON_Alarm : TON_TIME;
   END_VAR
BEGIN

   // Если давление ниже уставки в течерии 10 сек - выводим сигнал АВАРИЯ
   // 
   #TON_Alarm(IN := #DataPress.rInPress < #DataPress.rSetpoint, PT := t#10s);

   #DataPress.bAlarm_Press := #TON_Alarm.Q;
END_FUNCTION_BLOCK

FUNCTION_BLOCK "FB_SVETOFOR"   // FB19, SCL
{ S7_Optimized_Access := 'TRUE' }
VERSION : 0.1
   VAR_OUTPUT
      Зеленый : Bool;   // Включение зеленого света
      Желтый : Bool;   // Включение желтого
      Красный : Bool;   // красного
      Пищалка : Bool;
   END_VAR
   VAR
      AlarmPress : Bool;   // Авария по давлению
      bBezz_State : Bool;   // Состояние для выхода
      mAlarm : Bool;   // Сохранение сост АВАРИЯ
      mOpenWind : Bool;   // Сохранение сост Открыто Окно
      mPause : Bool;   // Сохранение сост Пауза
      mSterilFinish : Bool;
   END_VAR
BEGIN
   //Включение зеленого при старте конвейеров
   //
   IF "Разрешение работы конвейера" THEN
       #Зеленый := TRUE;
   ELSIF "bStartWork_Main_TunelPaster" AND NOT "Разрешение работы конвейера" THEN
       #Зеленый := "Time_2s";
   ELSE
       #Зеленый := FALSE;
   END_IF;

   // ___________________________________Упрвавление желтым сигналом________________________
   // 
   #Желтый := FALSE;
   IF "bOpenWindStartConveyor" OR "AlarmPress" OR ("iHMI_Num_StatrPaster" = 40) THEN
       #Желтый := TRUE;
   END_IF;
   IF "bStartWork_Sterilization" AND "bState_Stiril_Zone_OK" THEN
       #Желтый := TRUE;
   ELSIF "bStartWork_Sterilization" AND NOT "bState_Stiril_Zone_OK" THEN
       #Желтый := "Time_2s";
   END_IF;

   //______________________________________Управление карасным сигналом_____________________
   //
   #Красный := FALSE;
   IF "bMain_AlarmSystem" THEN
       #Красный := TRUE;
   END_IF;



   // __________________________________Управление пищалкой-______________________________
   // 
   ///По умолчанию отключаю пищалку
   #bBezz_State := FALSE;
   "RT_Alarm"(CLK:="bMain_AlarmSystem");


   //Условие включения звука при аварии
   IF "RT_Alarm".Q OR #mAlarm THEN
    //   #bBezz_State := TRUE;
       #mAlarm := TRUE;
   END_IF;

   //Условие включения при Вызове вспл окна оператора
   //
   "R_trig_OpenWindOper"(In := "bOpenWindStartConveyor");  //Триггер по открытию окна

   IF NOT "bOpenWindStartConveyor" THEN
       #mOpenWind := FALSE;    //Если окно закрыто - выкл звук

   ELSIF
       "R_trig_OpenWindOper".Q OR #mOpenWind AND NOT "bT_Alarm" THEN
       #mOpenWind := TRUE;

     //  #bBezz_State := "Time_1s";      //Включаем пищалку на цикл по 1 сек

   END_IF;


   // Условие включения при Паузе 
   // 
   "R_trig_Puasa"(In := ("iHMI_Num_StatrPaster" = 40));

   IF "iHMI_Num_StatrPaster" <> 40 THEN    //отключаем пищалку если не в состоянии Пауза
       #mPause := FALSE;
   ELSIF
       "R_trig_Puasa".Q OR #mPause AND NOT "bT_Alarm" THEN
       #mPause := TRUE;

      // #bBezz_State := "Time_1s";  //Включаем пищалку на цикл по 1 сек

   END_IF;

   //Условия для включения при стерилизации

   "RT_Steril_Finish"(CLK:="bHMI_Steril_Fimish");

   IF "RT_Steril_Finish".Q OR #mSterilFinish THEN
       #mSterilFinish := TRUE;
   END_IF;



   //Сбррос пищалки
   //
   IF "bZoomerOff" THEN
       #bBezz_State := FALSE;
       #mPause := FALSE;
       #mOpenWind := FALSE;
       #mAlarm := FALSE;
       #mSterilFinish := FALSE;
       ;
   END_IF;

   //Параметры для выхода на пищалку интенсивность
   IF #mAlarm THEN
       #bBezz_State := TRUE;
   ELSIF #mOpenWind THEN
       #bBezz_State := "Time_1s";
   ELSIF #mPause THEN
       #bBezz_State := "Time_0.5s";
   ELSIF #mSterilFinish THEN
       ;// #bBezz_State := "Time_2s";
   END_IF;

   //Присвоение значения на выход блока
   #Пищалка := #bBezz_State;

   //Вызов окна Операции стирилзации закончена

   "bOpenWindSterilFinish" := #mSterilFinish;
END_FUNCTION_BLOCK

FUNCTION_BLOCK "FB_Zone_Control_Steriliz"   // FB20, SCL
{ S7_Optimized_Access := 'FALSE' }
VERSION : 0.1
   VAR_INPUT
      bNewStart : Bool;   // Обнаружение нового старта, уставка без дельты
      DT_InParamZoneSteril : "Zone_Pararm";
   END_VAR
   VAR_OUTPUT
      ZoneStatusOut : "ZoneStatus";
      bInSetpoint : Bool;
      bOutOfRange : Bool;
      bHasPriority : Bool;
   END_VAR
   VAR
      R_Trig_Start : "R_trig";
      "#bNewStartCLic" : Bool;
      bSetpointReachedOnce : Bool;
   END_VAR
BEGIN
   // --- Сброс флага при необходимости ---
   // 
       //----Отслеживание нажания старта, по верхнему фронту-----
   #R_Trig_Start("In":= #bNewStart,Q => #"#bNewStartCLic");

   IF #"#bNewStartCLic" THEN
       #bSetpointReachedOnce := FALSE;
   END_IF;

   // --- Фиксация первого достижения уставки (точно или ±0.1) ---
   IF NOT #bSetpointReachedOnce AND ABS(#DT_InParamZoneSteril.rTemp - #DT_InParamZoneSteril.rSet) <= 1 THEN
       #bSetpointReachedOnce := TRUE;
   END_IF;

   // --- Расчёт попадания в уставку с учетом асимметричной дельты ---
   IF #bSetpointReachedOnce THEN
       #ZoneStatusOut.bInSetpoint := (#DT_InParamZoneSteril.rTemp >= (#DT_InParamZoneSteril.rSet - #DT_InParamZoneSteril.rDeltaDown)) AND
       (#DT_InParamZoneSteril.rTemp <= (#DT_InParamZoneSteril.rSet + #DT_InParamZoneSteril.rDeltaUP));
   ELSE
       // До первого достижения — строгое приближение (или узкая дельта)
       #ZoneStatusOut.bInSetpoint := ABS(#DT_InParamZoneSteril.rTemp - #DT_InParamZoneSteril.rSet) <= 1;
   END_IF;

   //Контроль зоны выхода из уставок значительно, греем снова до уставки до разрешения на старт

   IF (#DT_InParamZoneSteril.rTemp < (#DT_InParamZoneSteril.rSet - #DT_InParamZoneSteril.rDeltaDown)) OR
       (#DT_InParamZoneSteril.rTemp > (#DT_InParamZoneSteril.rSet + #DT_InParamZoneSteril.rDeltaUP)) THEN
       #bSetpointReachedOnce := FALSE;
   END_IF;


   // --- Остальные сигналы ---
   #ZoneStatusOut.bOutOfRange := NOT #ZoneStatusOut.bInSetpoint;
   #ZoneStatusOut.bHasPriority := #DT_InParamZoneSteril.bPriority;

   // Зеркалируем, если нужно
   #bInSetpoint := #ZoneStatusOut.bInSetpoint;
   #bOutOfRange := #ZoneStatusOut.bOutOfRange;
   #bHasPriority := #ZoneStatusOut.bHasPriority;
END_FUNCTION_BLOCK

FUNCTION_BLOCK "FB_Steril_Timer"   // FB22, SCL
{ S7_Optimized_Access := 'TRUE' }
VERSION : 0.1
   VAR_INPUT
      En_1 : Bool;   // Разрешение работы блока
      Start : Bool;   // Старт / Пауза
      SetTimeMin : Int;   // Уставка в минутах (задаётся с HMI)
   END_VAR
   VAR_OUTPUT
      RemainingMin : Int;   // Оставшиеся минуты
      RemainingSec : Int;   // Оставшиеся секунды
      TimeIsUp : Bool;   // Флаг конца времени
   END_VAR
   VAR
      TotalSec : DInt;   // Полное время в сек
      RemSec : DInt;   // Отсаток в сек
      bStartPrev : Bool;   // Для фронта
      bSecPulse : Bool;   // Секунда имп
      ton1 : TON_TIME;   // отсчет 1 сек
   END_VAR
BEGIN
   // ---------------------------------------------------------
   // Инициализация при EN = FALSE
   // ---------------------------------------------------------
   IF NOT #En_1 THEN
       #TotalSec := #SetTimeMin * 60;  // Пересчёт уставки в секунды
       #RemSec := #TotalSec;
       #RemainingMin := #SetTimeMin;
       #RemainingSec := 0;
       #TimeIsUp := FALSE;
       #ton1(IN := FALSE, PT := t#0s);
       RETURN;
   END_IF;

   // ---------------------------------------------------------
   // Генерация секундного импульса через TON (1 сек)
   // ---------------------------------------------------------
   #ton1(IN := #Start,
         PT := T#1S);

   IF #ton1.Q THEN
       #bSecPulse := TRUE;
       #ton1(IN := FALSE, PT := t#0s); // перезапуск таймера
   ELSE
       #bSecPulse := FALSE;
   END_IF;

   // ---------------------------------------------------------
   // Основная логика обратного отсчёта
   // ---------------------------------------------------------
   IF #Start AND (#RemSec > 0) THEN
       IF #bSecPulse THEN
           #RemSec := #RemSec - 1;
       END_IF;
   END_IF;

   // ---------------------------------------------------------
   // Если время вышло
   // ---------------------------------------------------------
   IF #RemSec <= 0 THEN
       #RemSec := 0;
       #TimeIsUp := TRUE;
   ELSE
       #TimeIsUp := FALSE;
   END_IF;

   // ---------------------------------------------------------
   // Преобразование остатка в минуты и секунды
   // ---------------------------------------------------------
   #RemainingMin := #RemSec / 60;
   #RemainingSec := #RemSec MOD 60;
END_FUNCTION_BLOCK

FUNCTION_BLOCK "FB_CheckZoneStatus"   // FB23, SCL
{ S7_Optimized_Access := 'FALSE' }
VERSION : 0.1
   VAR_OUTPUT
      bAllZones_Redy : Bool;   // Выход состояния всех зон ОК
      bPriority_Stop : Bool;   // Выход 1 - если есть метка остановки конвейера
      iZonesNumberFail : Int;   // ВЫход с Номером зоны
   END_VAR
   VAR
      aZoneS_Status : Array[1..7] of "ZoneStatus";   // Массив с данными по всем зонам
      i : Int;
      AllZone_Ok : Bool;   // Состояние всех зон ОК
      HaveStopPriority : Bool;   // В зоне есть метка для остановки конвейера
      iNumber : Int;   // Номер зоны, где отклонение температуры
   END_VAR
BEGIN

   //Что бы не контролировал готовность зоны 4 ее не надо контролировать
   //"ЗОНЫ_Параметры".Zone_4.bOUT_ZoneStatus.bInSetpoint := TRUE;
   //-------------------------------------------------------------------------------------------//
   //
           // ----Сбор данных по всем зонам в массив для обработки-----
           #aZoneS_Status[1] := "ЗОНЫ_Параметры".Zone_1.bOUT_ZoneStatus;
           #aZoneS_Status[2] := "ЗОНЫ_Параметры".Zone_2.bOUT_ZoneStatus;
           #aZoneS_Status[3] := "ЗОНЫ_Параметры".Zone_3.bOUT_ZoneStatus;
           #aZoneS_Status[4] := "ЗОНЫ_Параметры".Zone_4.bOUT_ZoneStatus;
           #aZoneS_Status[5] := "ЗОНЫ_Параметры".Zone_5.bOUT_ZoneStatus;
           #aZoneS_Status[6] := "ЗОНЫ_Параметры".Zone_6.bOUT_ZoneStatus;
           #aZoneS_Status[7] := "ЗОНЫ_Параметры".Zone_7.bOUT_ZoneStatus;


           //Сброс маркеров по умолчанию----
   #AllZone_Ok := TRUE;    
   #HaveStopPriority := FALSE;
   #iNumber := 0;
              // ----Цикл для перебора всех зон значение выставить по количеству зон----
   FOR #i := 1 TO 7 DO
       IF (#i = 5 OR #i = 6) THEN  //Пропускаем статусы зон
           CONTINUE;
           ;
       END_IF;
       IF NOT #aZoneS_Status[#i].bInSetpoint THEN
           #AllZone_Ok := FALSE;
           #iNumber := #i;
           IF #aZoneS_Status[#i].bHasPriority THEN
               #HaveStopPriority := TRUE;
           END_IF;
       END_IF;
   END_FOR;

   /// Присвоение переменных к выходам
   #bAllZones_Redy := #AllZone_Ok;
   #bPriority_Stop := #HaveStopPriority;
   #iZonesNumberFail := #iNumber;
END_FUNCTION_BLOCK

FUNCTION_BLOCK "Test_Beep"   // FB24, SCL
{ S7_Optimized_Access := 'TRUE' }
VERSION : 0.1
   VAR
      BzzzState : Bool;
      mOpWind : Bool;
      mPause : Bool;
      mAlarm : Bool;
   END_VAR
BEGIN
   #BzzzState := FALSE;
   //Условие включения звука при аварии
   IF "bT_Alarm" OR #mAlarm THEN
      // #BzzzState := TRUE;
       #mAlarm := TRUE;
   END_IF;

   //Условие включения при Вызове вспл окна оператора
   //
   "R_TRIG_TestOpenWind"(CLK:="bTOpenWind");
   IF NOT "bTOpenWind" THEN
       #mOpWind := FALSE;

   ELSIF
       "R_TRIG_TestOpenWind".Q OR #mOpWind AND NOT "bT_Alarm" THEN
      // #BzzzState := "Time_0.5s";
       #mOpWind := TRUE;
   END_IF;



   // Условие включения при Паузе 
   // 
   "R_TRIG_TestPause"(CLK:=("iTestPause" = 40));


   IF "iTestPause" <> 40 THEN
       #mPause := FALSE;
   ELSIF
       "R_TRIG_TestPause".Q OR #mPause AND NOT "bT_Alarm" THEN
       //#BzzzState := "Time_0.2s";
       #mPause := TRUE;
   END_IF;
   ;

   //Сбррос пищалки
   //
   IF "bTZoomOff" THEN
       #BzzzState := FALSE;
       #mPause := FALSE;
       #mOpWind := FALSE;
       #mAlarm := FALSE;
       ;
   END_IF;

   IF #mAlarm THEN
       #BzzzState := TRUE;
   ELSIF #mOpWind THEN
       #BzzzState := "Time_1s";
   ELSIF #mPause THEN
       #BzzzState := "Time_0.5s";
   END_IF;
END_FUNCTION_BLOCK

FUNCTION_BLOCK "FB_Mode_STIRIL"   // FB25, SCL
{ S7_Optimized_Access := 'TRUE' }
VERSION : 0.1
   VAR_INPUT
      bEn_Mode : Bool;   // разрешение на работу
   END_VAR
BEGIN
   IF NOT #bEn_Mode THEN
       RETURN;
   END_IF;

   IF #bEn_Mode THEN
       //Открываем калпана запорные
       "FVs_o/p".FV_2.bOpenCmd := TRUE;    //Клапан пара
       "FVs_o/p".FV_3.bOpenCmd := TRUE;    //Клапан Стерилизации

       //Открываем клапана регулирующие
       "FVs_Regul".FV_Regul_1."bAutoOpen/Close" := TRUE;
       "FVs_Regul".FV_Regul_2."bAutoOpen/Close" := TRUE;
       "FVs_Regul".FV_Regul_3."bAutoOpen/Close" := TRUE;
       "FVs_Regul".FV_Regul_4."bAutoOpen/Close" := TRUE;
       "FVs_Regul".FV_Regul_7."bAutoOpen/Close" := TRUE;


       //Передача уставки для пид регуляторов
       //
       "DB2_HMI_SET".k_PID_Zona1.Set := "Зоны_Стерилизации_Парам"."Steril_Zona-1".rSet;
       "DB2_HMI_SET".k_PID_Zona2.Set := "Зоны_Стерилизации_Парам"."Steril_Zona-2".rSet;
       "DB2_HMI_SET".k_PID_Zona3.Set := "Зоны_Стерилизации_Парам"."Steril_Zona-3".rSet;
       "DB2_HMI_SET".k_PID_Zona4.Set := "Зоны_Стерилизации_Парам"."Steril_Zona-4".rSet;
       "DB2_HMI_SET".k_PID_Zona7.Set := "Зоны_Стерилизации_Парам"."Steril_Zona-7".rSet;
       ;


       //Старт насосов
       //
       "Pumps".Pump_1.bAutoMode_Work := TRUE;
       "Pumps".Pump_2.bAutoMode_Work := TRUE;
       "Pumps".Pump_3.bAutoMode_Work := TRUE;
       "Pumps".Pump_4.bAutoMode_Work := TRUE;
       "Pumps".Pump_5.bAutoMode_Work := TRUE;
       "Pumps".Pump_6.bAutoMode_Work := TRUE;
       "Pumps".Pump_7.bAutoMode_Work := TRUE;




   END_IF;
END_FUNCTION_BLOCK

FUNCTION_BLOCK "FB_Mode_Paster"   // FB26, SCL
{ S7_Optimized_Access := 'TRUE' }
VERSION : 0.1
   VAR_INPUT
      bEn_Mode : Bool;   // разрешение на работу
   END_VAR
BEGIN
   IF NOT #bEn_Mode THEN
       RETURN;
   END_IF;

   IF #bEn_Mode THEN
       //Открываем калпана запорные
       "FVs_o/p".FV_2.bOpenCmd := TRUE;    //Клапан пара
       "FVs_o/p".FV_3.bOpenCmd := FALSE;    //Клапан Стерилизации

       //Открываем клапана регулирующие
       "FVs_Regul".FV_Regul_1."bAutoOpen/Close" := TRUE;
       "FVs_Regul".FV_Regul_2."bAutoOpen/Close" := TRUE;
       "FVs_Regul".FV_Regul_3."bAutoOpen/Close" := TRUE;
       "FVs_Regul".FV_Regul_4."bAutoOpen/Close" := TRUE;
       "FVs_Regul".FV_Regul_7."bAutoOpen/Close" := TRUE;


       //Старт насосов
       //
       "Pumps".Pump_1.bAutoMode_Work := TRUE;
       "Pumps".Pump_2.bAutoMode_Work := TRUE;
       "Pumps".Pump_3.bAutoMode_Work := TRUE;
       "Pumps".Pump_4.bAutoMode_Work := TRUE;
       "Pumps".Pump_5.bAutoMode_Work := TRUE;
       "Pumps".Pump_6.bAutoMode_Work := TRUE;
       "Pumps".Pump_7.bAutoMode_Work := TRUE;

       //Передача уставки для пид регуляторов
       //
       "DB2_HMI_SET".k_PID_Zona1.Set := "ЗОНЫ_Параметры".Zone_1.rSet;
       "DB2_HMI_SET".k_PID_Zona2.Set := "ЗОНЫ_Параметры".Zone_2.rSet;
       "DB2_HMI_SET".k_PID_Zona3.Set := "ЗОНЫ_Параметры".Zone_3.rSet;
       "DB2_HMI_SET".k_PID_Zona4.Set := "ЗОНЫ_Параметры".Zone_4.rSet;
       "DB2_HMI_SET".k_PID_Zona7.Set := "ЗОНЫ_Параметры".Zone_7.rSet;
       ;


   END_IF;
END_FUNCTION_BLOCK

FUNCTION "Клапана_О/З" : Void   // FC1, LAD
{ S7_Optimized_Access := 'TRUE' }
VERSION : 0.1
BEGIN

REGION Network 1: FV-1
   // Клапан подпитки емкости водой
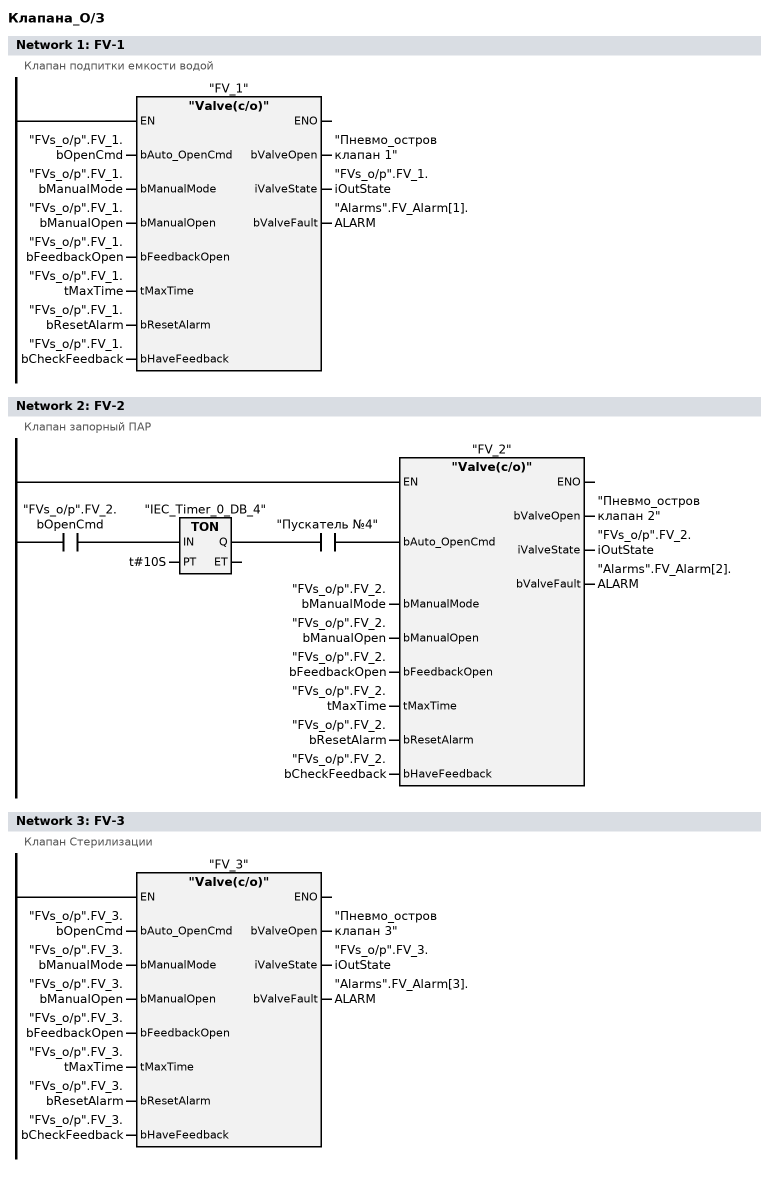
   RUNG wire#powerrail
      "FV_1"(bAuto_OpenCmd := "FVs_o/p".FV_1.bOpenCmd, bManualMode := "FVs_o/p".FV_1.bManualMode, bManualOpen := "FVs_o/p".FV_1.bManualOpen, bFeedbackOpen := "FVs_o/p".FV_1.bFeedbackOpen, tMaxTime := "FVs_o/p".FV_1.tMaxTime, bResetAlarm := "FVs_o/p".FV_1.bResetAlarm, bHaveFeedback := "FVs_o/p".FV_1.bCheckFeedback, bValveOpen => "Пневмо_остров клапан 1", iValveState => "FVs_o/p".FV_1.iOutState, bValveFault => "Alarms".FV_Alarm[1].ALARM)
   END_RUNG
   // the same network as SCL:
   "FV_1"(bAuto_OpenCmd := "FVs_o/p".FV_1.bOpenCmd,   // "Valve(c/o)"
          bManualMode := "FVs_o/p".FV_1.bManualMode,
          bManualOpen := "FVs_o/p".FV_1.bManualOpen,
          bFeedbackOpen := "FVs_o/p".FV_1.bFeedbackOpen,
          tMaxTime := "FVs_o/p".FV_1.tMaxTime,
          bResetAlarm := "FVs_o/p".FV_1.bResetAlarm,
          bHaveFeedback := "FVs_o/p".FV_1.bCheckFeedback,
          bValveOpen => "Пневмо_остров клапан 1",
          iValveState => "FVs_o/p".FV_1.iOutState,
          bValveFault => "Alarms".FV_Alarm[1].ALARM);
END_REGION

REGION Network 2: FV-2
   // Клапан запорный ПАР
   "IEC_Timer_0_DB_4".TON(IN := "FVs_o/p".FV_2.bOpenCmd, PT := t#10S);
   "FV_2"(bAuto_OpenCmd := "IEC_Timer_0_DB_4".Q AND "Пускатель №4",   // "Valve(c/o)"
          bManualMode := "FVs_o/p".FV_2.bManualMode,
          bManualOpen := "FVs_o/p".FV_2.bManualOpen,
          bFeedbackOpen := "FVs_o/p".FV_2.bFeedbackOpen,
          tMaxTime := "FVs_o/p".FV_2.tMaxTime,
          bResetAlarm := "FVs_o/p".FV_2.bResetAlarm,
          bHaveFeedback := "FVs_o/p".FV_2.bCheckFeedback,
          bValveOpen => "Пневмо_остров клапан 2",
          iValveState => "FVs_o/p".FV_2.iOutState,
          bValveFault => "Alarms".FV_Alarm[2].ALARM);
END_REGION

REGION Network 3: FV-3
   // Клапан Стерилизации
   RUNG wire#powerrail
      "FV_3"(bAuto_OpenCmd := "FVs_o/p".FV_3.bOpenCmd, bManualMode := "FVs_o/p".FV_3.bManualMode, bManualOpen := "FVs_o/p".FV_3.bManualOpen, bFeedbackOpen := "FVs_o/p".FV_3.bFeedbackOpen, tMaxTime := "FVs_o/p".FV_3.tMaxTime, bResetAlarm := "FVs_o/p".FV_3.bResetAlarm, bHaveFeedback := "FVs_o/p".FV_3.bCheckFeedback, bValveOpen => "Пневмо_остров клапан 3", iValveState => "FVs_o/p".FV_3.iOutState, bValveFault => "Alarms".FV_Alarm[3].ALARM)
   END_RUNG
   // the same network as SCL:
   "FV_3"(bAuto_OpenCmd := "FVs_o/p".FV_3.bOpenCmd,   // "Valve(c/o)"
          bManualMode := "FVs_o/p".FV_3.bManualMode,
          bManualOpen := "FVs_o/p".FV_3.bManualOpen,
          bFeedbackOpen := "FVs_o/p".FV_3.bFeedbackOpen,
          tMaxTime := "FVs_o/p".FV_3.tMaxTime,
          bResetAlarm := "FVs_o/p".FV_3.bResetAlarm,
          bHaveFeedback := "FVs_o/p".FV_3.bCheckFeedback,
          bValveOpen => "Пневмо_остров клапан 3",
          iValveState => "FVs_o/p".FV_3.iOutState,
          bValveFault => "Alarms".FV_Alarm[3].ALARM);
END_REGION
END_FUNCTION

FUNCTION "Клапана_Регул" : Void   // FC2, LAD
{ S7_Optimized_Access := 'TRUE' }
VERSION : 0.1
BEGIN

